LIN {X -0.135,Y -641.300,Z 780.617,A 0.000,B 0.000,C 90.000,E1 327.041} C_DIS
LIN {X 0.233,Y -645.781,Z 780.611,A 0.000,B 0.000,C 90.000,E1 326.008} C_DIS
LIN {X 0.128,Y -649.952,Z 780.606,A 0.000,B 0.000,C 90.000,E1 325.022} C_DIS
LIN {X 0.080,Y -653.850,Z 780.600,A 0.000,B 0.000,C 90.000,E1 324.036} C_DIS
LIN {X 0.081,Y -657.396,Z 780.595,A 0.000,B 0.000,C 90.000,E1 323.050} C_DIS
LIN {X 0.118,Y -660.884,Z 780.589,A 0.000,B 0.000,C 90.000,E1 322.065} C_DIS
LIN {X -0.359,Y -664.827,Z 780.583,A 0.000,B 0.000,C 90.000,E1 320.884} C_DIS
LIN {X -0.338,Y -667.859,Z 780.577,A 0.000,B 0.000,C 90.000,E1 319.908} C_DIS
LIN {X -0.271,Y -671.350,Z 780.570,A 0.000,B 0.000,C 90.000,E1 318.690} C_DIS
LIN {X -0.147,Y -674.584,Z 780.564,A 0.000,B 0.000,C 90.000,E1 317.472} C_DIS
LIN {X -0.008,Y -677.297,Z 780.557,A 0.000,B 0.000,C 90.000,E1 316.257} C_DIS
LIN {X -0.291,Y -679.717,Z 780.550,A 0.000,B 0.000,C 90.000,E1 315.081} C_DIS
LIN {X -0.066,Y -681.929,Z 780.544,A 0.000,B 0.000,C 90.000,E1 313.866} C_DIS
LIN {X -0.279,Y -683.940,Z 780.537,A 0.000,B 0.000,C 90.000,E1 312.690} C_DIS
LIN {X 0.049,Y -685.760,Z 780.530,A 0.000,B 0.000,C 90.000,E1 311.472} C_DIS
LIN {X -0.114,Y -687.422,Z 780.524,A 0.000,B 0.000,C 90.000,E1 310.297} C_DIS
LIN {X -0.180,Y -688.753,Z 780.517,A 0.000,B 0.000,C 90.000,E1 309.116} C_DIS
LIN {X -0.050,Y -690.190,Z 780.509,A 0.000,B 0.000,C 90.000,E1 307.684} C_DIS
LIN {X -0.124,Y -691.112,Z 780.504,A 0.000,B 0.000,C 90.000,E1 306.744} C_DIS
LIN {X 0.057,Y -692.345,Z 780.496,A 0.000,B 0.000,C 90.000,E1 305.311} C_DIS
LIN {X 0.205,Y -693.268,Z 780.490,A 0.000,B 0.000,C 90.000,E1 304.119} C_DIS
LIN {X 0.235,Y -694.476,Z 780.481,A 0.000,B 0.000,C 90.000,E1 302.467} C_DIS
LIN {X -0.090,Y -695.755,Z 780.471,A 0.000,B 0.000,C 90.000,E1 300.846} C_DIS
LIN {X 0.307,Y -696.373,Z 780.466,A 0.000,B 0.000,C 90.000,E1 299.873} C_DIS
LIN {X 0.018,Y -697.038,Z 780.458,A 0.000,B 0.000,C 90.000,E1 298.487} C_DIS
LIN {X -0.332,Y -697.783,Z 780.449,A 0.000,B 0.000,C 90.000,E1 296.873} C_DIS
LIN {X 0.192,Y -699.103,Z 780.437,A 0.000,B 0.000,C 90.000,E1 294.719} C_DIS
LIN {X 0.088,Y -699.011,Z 780.435,A 0.000,B 0.000,C 90.000,E1 294.259} C_DIS
LIN {X 0.067,Y -698.774,Z 780.434,A 0.000,B 0.000,C 90.000,E1 294.027} C_DIS
LIN {X -0.045,Y -697.662,Z 780.431,A 0.000,B 0.000,C 90.000,E1 293.567} C_DIS
LIN {X -0.062,Y -696.673,Z 780.430,A 0.000,B 0.000,C 90.000,E1 293.334} C_DIS
LIN {X 0.195,Y -694.685,Z 780.428,A 0.000,B 0.000,C 90.000,E1 293.078} C_DIS
LIN {X 0.174,Y -692.575,Z 780.427,A 0.000,B 0.000,C 90.000,E1 292.845} C_DIS
LIN {X -0.344,Y -691.398,Z 780.426,A 0.000,B 0.000,C 90.000,E1 292.770} C_DIS
LIN {X -0.222,Y -689.693,Z 780.426,A 0.000,B 0.000,C 90.000,E1 292.642} C_DIS
LIN {X 0.320,Y -683.390,Z 780.424,A 0.000,B 0.000,C 90.000,E1 292.333} C_DIS
LIN {X 0.365,Y -679.497,Z 780.424,A 0.000,B 0.000,C 90.000,E1 292.206} C_DIS
LIN {X 0.119,Y -673.718,Z 780.423,A 0.000,B 0.000,C 90.000,E1 292.078} C_DIS
LIN {X -0.079,Y -664.421,Z 780.422,A 0.000,B 0.000,C 90.000,E1 291.950} C_DIS
LIN {X 0.178,Y -654.094,Z 780.421,A 0.000,B 0.000,C 90.000,E1 291.770} C_DIS
LIN {X 0.001,Y -640.328,Z 780.420,A 0.000,B 0.000,C 90.000,E1 291.535} C_DIS
LIN {X 0.328,Y -616.048,Z 780.417,A 0.000,B 0.000,C 90.000,E1 290.972} C_DIS
LIN {X -0.071,Y -595.435,Z 780.414,A 0.000,B 0.000,C 90.000,E1 290.482} C_DIS
LIN {X -0.040,Y -571.555,Z 780.410,A 0.000,B 0.000,C 90.000,E1 289.758} C_DIS
LIN {X 0.063,Y -565.181,Z 780.409,A 0.000,B 0.000,C 90.000,E1 289.523} C_DIS
LIN {X 0.046,Y -560.669,Z 780.407,A 0.000,B 0.000,C 90.000,E1 289.322} C_DIS
LIN {X -0.169,Y -557.657,Z 780.406,A 0.000,B 0.000,C 90.000,E1 289.087} C_DIS
LIN {X -0.152,Y -556.753,Z 780.405,A 0.000,B 0.000,C 90.000,E1 288.906} C_DIS
LIN {X 0.258,Y -556.190,Z 780.404,A 0.000,B 0.000,C 90.000,E1 288.725} C_DIS
LIN {X -0.274,Y -555.270,Z 780.402,A 0.000,B 0.000,C 90.000,E1 288.362} C_DIS
LIN {X 0.220,Y -554.706,Z 780.399,A 0.000,B 0.000,C 90.000,E1 287.764} C_DIS
LIN {X -0.169,Y -554.398,Z 780.394,A 0.000,B 0.000,C 90.000,E1 286.968} C_DIS
LIN {X 0.001,Y -553.355,Z 780.382,A 0.000,B 0.000,C 90.000,E1 284.717} C_DIS
LIN {X -0.097,Y -552.709,Z 780.371,A 0.000,B 0.000,C 90.000,E1 282.771} C_DIS
LIN {X 0.209,Y -551.975,Z 780.360,A 0.000,B 0.000,C 90.000,E1 280.782} C_DIS
LIN {X 0.251,Y -551.570,Z 780.352,A 0.000,B 0.000,C 90.000,E1 279.378} C_DIS
LIN {X -0.222,Y -551.091,Z 780.341,A 0.000,B 0.000,C 90.000,E1 277.466} C_DIS
LIN {X -0.037,Y -550.765,Z 780.337,A 0.000,B 0.000,C 90.000,E1 276.606} C_DIS
LIN {X -0.194,Y -549.990,Z 780.329,A 0.000,B 0.000,C 90.000,E1 275.220} C_DIS
LIN {X 0.172,Y -548.872,Z 780.320,A 0.000,B 0.000,C 90.000,E1 273.498} C_DIS
LIN {X 0.007,Y -547.653,Z 780.309,A 0.000,B 0.000,C 90.000,E1 271.547} C_DIS
LIN {X 0.192,Y -546.992,Z 780.302,A 0.000,B 0.000,C 90.000,E1 270.401} C_DIS
LIN {X -0.093,Y -545.804,Z 780.293,A 0.000,B 0.000,C 90.000,E1 268.740} C_DIS
LIN {X 0.211,Y -544.440,Z 780.282,A 0.000,B 0.000,C 90.000,E1 266.731} C_DIS
LIN {X -0.058,Y -543.288,Z 780.271,A 0.000,B 0.000,C 90.000,E1 264.780} C_DIS
LIN {X 0.118,Y -542.505,Z 780.265,A 0.000,B 0.000,C 90.000,E1 263.628} C_DIS
LIN {X -0.188,Y -541.619,Z 780.258,A 0.000,B 0.000,C 90.000,E1 262.527} C_DIS
LIN {X 0.159,Y -539.693,Z 780.246,A 0.000,B 0.000,C 90.000,E1 260.218} C_DIS
LIN {X -0.021,Y -538.448,Z 780.238,A 0.000,B 0.000,C 90.000,E1 258.814} C_DIS
LIN {X -0.218,Y -537.131,Z 780.230,A 0.000,B 0.000,C 90.000,E1 257.409} C_DIS
LIN {X 0.204,Y -535.771,Z 780.222,A 0.000,B 0.000,C 90.000,E1 255.936} C_DIS
LIN {X 0.076,Y -534.243,Z 780.214,A 0.000,B 0.000,C 90.000,E1 254.519} C_DIS
LIN {X -0.040,Y -531.633,Z 780.201,A 0.000,B 0.000,C 90.000,E1 252.236} C_DIS
LIN {X 0.062,Y -529.928,Z 780.193,A 0.000,B 0.000,C 90.000,E1 250.786} C_DIS
LIN {X -0.057,Y -528.729,Z 780.189,A 0.000,B 0.000,C 90.000,E1 249.934} C_DIS
LIN {X -0.169,Y -525.843,Z 780.177,A 0.000,B 0.000,C 90.000,E1 247.922} C_DIS
LIN {X 0.025,Y -522.729,Z 780.166,A 0.000,B 0.000,C 90.000,E1 245.869} C_DIS
LIN {X 0.231,Y -521.360,Z 780.161,A 0.000,B 0.000,C 90.000,E1 244.973} C_DIS
LIN {X 0.044,Y -518.031,Z 780.150,A 0.000,B 0.000,C 90.000,E1 242.948} C_DIS
LIN {X 0.103,Y -515.939,Z 780.143,A 0.000,B 0.000,C 90.000,E1 241.769} C_DIS
LIN {X 0.136,Y -513.734,Z 780.137,A 0.000,B 0.000,C 90.000,E1 240.589} C_DIS
LIN {X 0.039,Y -510.898,Z 780.129,A 0.000,B 0.000,C 90.000,E1 239.125} C_DIS
LIN {X -0.012,Y -508.599,Z 780.122,A 0.000,B 0.000,C 90.000,E1 237.946} C_DIS
LIN {X 0.011,Y -506.111,Z 780.115,A 0.000,B 0.000,C 90.000,E1 236.755} C_DIS
LIN {X -0.165,Y -504.204,Z 780.110,A 0.000,B 0.000,C 90.000,E1 235.881} C_DIS
LIN {X -0.195,Y -501.477,Z 780.104,A 0.000,B 0.000,C 90.000,E1 234.689} C_DIS
LIN {X -0.267,Y -498.555,Z 780.097,A 0.000,B 0.000,C 90.000,E1 233.497} C_DIS
LIN {X -0.224,Y -494.759,Z 780.089,A 0.000,B 0.000,C 90.000,E1 231.984} C_DIS
LIN {X -0.103,Y -490.281,Z 780.079,A 0.000,B 0.000,C 90.000,E1 230.150} C_DIS
LIN {X -0.037,Y -484.029,Z 780.063,A 0.000,B 0.000,C 90.000,E1 227.391} C_DIS
LIN {X 0.308,Y -480.729,Z 780.055,A 0.000,B 0.000,C 90.000,E1 225.810} C_DIS
LIN {X -0.314,Y -476.642,Z 780.044,A 0.000,B 0.000,C 90.000,E1 224.028} C_DIS
LIN {X -0.110,Y -473.271,Z 780.036,A 0.000,B 0.000,C 90.000,E1 222.447} C_DIS
LIN {X 0.139,Y -469.135,Z 780.025,A 0.000,B 0.000,C 90.000,E1 220.539} C_DIS
LIN {X -0.014,Y -465.253,Z 780.015,A 0.000,B 0.000,C 90.000,E1 218.669} C_DIS
LIN {X -0.049,Y -459.917,Z 780.001,A 0.000,B 0.000,C 90.000,E1 216.137} C_DIS
LIN {X 0.133,Y -455.957,Z 779.990,A 0.000,B 0.000,C 90.000,E1 214.199} C_DIS
LIN {X 0.074,Y -451.441,Z 779.978,A 0.000,B 0.000,C 90.000,E1 211.957} C_DIS
LIN {X 0.120,Y -448.322,Z 779.969,A 0.000,B 0.000,C 90.000,E1 210.335} C_DIS
LIN {X -0.129,Y -445.213,Z 779.960,A 0.000,B 0.000,C 90.000,E1 208.743} C_DIS
LIN {X 0.132,Y -442.126,Z 779.951,A 0.000,B 0.000,C 90.000,E1 207.078} C_DIS
LIN {X -0.058,Y -438.986,Z 779.941,A 0.000,B 0.000,C 90.000,E1 205.463} C_DIS
LIN {X -0.111,Y -435.916,Z 779.932,A 0.000,B 0.000,C 90.000,E1 203.823} C_DIS
LIN {X 0.003,Y -432.784,Z 779.923,A 0.000,B 0.000,C 90.000,E1 202.153} C_DIS
LIN {X 0.243,Y -430.223,Z 779.916,A 0.000,B 0.000,C 90.000,E1 200.791} C_DIS
LIN {X -0.052,Y -425.741,Z 779.903,A 0.000,B 0.000,C 90.000,E1 198.489} C_DIS
LIN {X -0.025,Y -422.562,Z 779.893,A 0.000,B 0.000,C 90.000,E1 196.804} C_DIS
LIN {X -0.183,Y -419.202,Z 779.884,A 0.000,B 0.000,C 90.000,E1 195.134} C_DIS
LIN {X 0.087,Y -414.754,Z 779.871,A 0.000,B 0.000,C 90.000,E1 192.715} C_DIS
LIN {X 0.062,Y -411.612,Z 779.861,A 0.000,B 0.000,C 90.000,E1 191.007} C_DIS
LIN {X -0.145,Y -407.322,Z 779.848,A 0.000,B 0.000,C 90.000,E1 188.624} C_DIS
LIN {X -0.144,Y -405.096,Z 779.840,A 0.000,B 0.000,C 90.000,E1 187.239} C_DIS
LIN {X 0.178,Y -402.144,Z 779.831,A 0.000,B 0.000,C 90.000,E1 185.454} C_DIS
LIN {X 0.078,Y -395.784,Z 779.807,A 0.000,B 0.000,C 90.000,E1 181.260} C_DIS
LIN {X 0.077,Y -393.265,Z 779.795,A 0.000,B 0.000,C 90.000,E1 179.141} C_DIS
LIN {X -0.127,Y -390.209,Z 779.780,A 0.000,B 0.000,C 90.000,E1 176.331} C_DIS
LIN {X -0.108,Y -388.525,Z 779.770,A 0.000,B 0.000,C 90.000,E1 174.546} C_DIS
LIN {X 0.128,Y -386.230,Z 779.756,A 0.000,B 0.000,C 90.000,E1 172.008} C_DIS
LIN {X 0.022,Y -384.179,Z 779.742,A 0.000,B 0.000,C 90.000,E1 169.511} C_DIS
LIN {X 0.000,Y -382.678,Z 779.730,A 0.000,B 0.000,C 90.000,E1 167.353} C_DIS
LIN {X 0.105,Y -381.329,Z 779.716,A 0.000,B 0.000,C 90.000,E1 164.810} C_DIS
LIN {X 0.012,Y -380.680,Z 779.708,A 0.000,B 0.000,C 90.000,E1 163.378} C_DIS
LIN {X 0.027,Y -379.601,Z 779.690,A 0.000,B 0.000,C 90.000,E1 160.115} C_DIS
LIN {X -0.068,Y -379.365,Z 779.661,A 0.000,B 0.000,C 90.000,E1 155.049} C_DIS
LIN {X -0.006,Y -380.951,Z 779.639,A 0.000,B 0.000,C 90.000,E1 151.051} C_DIS
LIN {X -0.102,Y -383.270,Z 779.625,A 0.000,B 0.000,C 90.000,E1 148.535} C_DIS
LIN {X -0.105,Y -384.702,Z 779.619,A 0.000,B 0.000,C 90.000,E1 147.454} C_DIS
LIN {X -0.161,Y -388.401,Z 779.607,A 0.000,B 0.000,C 90.000,E1 145.308} C_DIS
LIN {X 0.051,Y -390.026,Z 779.603,A 0.000,B 0.000,C 90.000,E1 144.562} C_DIS
LIN {X -0.046,Y -392.045,Z 779.599,A 0.000,B 0.000,C 90.000,E1 143.863} C_DIS
LIN {X 0.108,Y -394.435,Z 779.595,A 0.000,B 0.000,C 90.000,E1 143.130} C_DIS
LIN {X 0.179,Y -397.031,Z 779.592,A 0.000,B 0.000,C 90.000,E1 142.477} C_DIS
LIN {X 0.041,Y -399.851,Z 779.588,A 0.000,B 0.000,C 90.000,E1 141.904} C_DIS
LIN {X 0.055,Y -402.995,Z 779.586,A 0.000,B 0.000,C 90.000,E1 141.376} C_DIS
LIN {X -0.179,Y -407.195,Z 779.582,A 0.000,B 0.000,C 90.000,E1 140.803} C_DIS
LIN {X -0.022,Y -422.989,Z 779.572,A 0.000,B 0.000,C 90.000,E1 138.895} C_DIS
LIN {X -0.088,Y -439.732,Z 779.561,A 0.000,B 0.000,C 90.000,E1 137.067} C_DIS
LIN {X 0.241,Y -449.355,Z 779.556,A 0.000,B 0.000,C 90.000,E1 135.972} C_DIS
LIN {X 0.037,Y -458.769,Z 779.550,A 0.000,B 0.000,C 90.000,E1 134.919} C_DIS
LIN {X 0.196,Y -465.141,Z 779.545,A 0.000,B 0.000,C 90.000,E1 134.109} C_DIS
LIN {X -0.046,Y -473.687,Z 779.539,A 0.000,B 0.000,C 90.000,E1 133.056} C_DIS
LIN {X -0.070,Y -480.870,Z 779.534,A 0.000,B 0.000,C 90.000,E1 132.123} C_DIS
LIN {X -0.026,Y -486.422,Z 779.530,A 0.000,B 0.000,C 90.000,E1 131.353} C_DIS
LIN {X -0.229,Y -492.767,Z 779.525,A 0.000,B 0.000,C 90.000,E1 130.458} C_DIS
LIN {X 0.252,Y -497.825,Z 779.520,A 0.000,B 0.000,C 90.000,E1 129.644} C_DIS
LIN {X -0.013,Y -501.651,Z 779.517,A 0.000,B 0.000,C 90.000,E1 129.072} C_DIS
LIN {X -0.147,Y -508.748,Z 779.510,A 0.000,B 0.000,C 90.000,E1 127.890} C_DIS
LIN {X -0.221,Y -512.922,Z 779.506,A 0.000,B 0.000,C 90.000,E1 127.156} C_DIS
LIN {X -0.032,Y -517.651,Z 779.501,A 0.000,B 0.000,C 90.000,E1 126.251} C_DIS
LIN {X -0.079,Y -522.953,Z 779.496,A 0.000,B 0.000,C 90.000,E1 125.231} C_DIS
LIN {X 0.263,Y -525.864,Z 779.492,A 0.000,B 0.000,C 90.000,E1 124.612} C_DIS
LIN {X 0.061,Y -527.701,Z 779.490,A 0.000,B 0.000,C 90.000,E1 124.199} C_DIS
LIN {X -0.095,Y -530.217,Z 779.487,A 0.000,B 0.000,C 90.000,E1 123.658} C_DIS
LIN {X 0.293,Y -533.847,Z 779.482,A 0.000,B 0.000,C 90.000,E1 122.752} C_DIS
LIN {X -0.317,Y -538.451,Z 779.476,A 0.000,B 0.000,C 90.000,E1 121.671} C_DIS
LIN {X -0.133,Y -541.646,Z 779.471,A 0.000,B 0.000,C 90.000,E1 120.797} C_DIS
LIN {X 0.084,Y -544.591,Z 779.466,A 0.000,B 0.000,C 90.000,E1 119.922} C_DIS
LIN {X -0.187,Y -548.316,Z 779.460,A 0.000,B 0.000,C 90.000,E1 118.821} C_DIS
LIN {X -0.165,Y -550.955,Z 779.455,A 0.000,B 0.000,C 90.000,E1 117.975} C_DIS
LIN {X -0.116,Y -553.416,Z 779.451,A 0.000,B 0.000,C 90.000,E1 117.129} C_DIS
LIN {X -0.046,Y -555.467,Z 779.446,A 0.000,B 0.000,C 90.000,E1 116.283} C_DIS
LIN {X -0.200,Y -557.174,Z 779.441,A 0.000,B 0.000,C 90.000,E1 115.463} C_DIS
LIN {X 0.174,Y -558.623,Z 779.437,A 0.000,B 0.000,C 90.000,E1 114.591} C_DIS
LIN {X 0.057,Y -559.762,Z 779.432,A 0.000,B 0.000,C 90.000,E1 113.770} C_DIS
LIN {X -0.052,Y -561.988,Z 779.421,A 0.000,B 0.000,C 90.000,E1 111.844} C_DIS
LIN {X -0.032,Y -563.169,Z 779.415,A 0.000,B 0.000,C 90.000,E1 110.737} C_DIS
LIN {X 0.138,Y -564.459,Z 779.408,A 0.000,B 0.000,C 90.000,E1 109.341} C_DIS
LIN {X 0.182,Y -565.400,Z 779.401,A 0.000,B 0.000,C 90.000,E1 108.236} C_DIS
LIN {X -0.174,Y -566.633,Z 779.392,A 0.000,B 0.000,C 90.000,E1 106.622} C_DIS
LIN {X 0.044,Y -567.863,Z 779.383,A 0.000,B 0.000,C 90.000,E1 104.954} C_DIS
LIN {X -0.230,Y -569.434,Z 779.372,A 0.000,B 0.000,C 90.000,E1 103.063} C_DIS
LIN {X -0.038,Y -571.056,Z 779.362,A 0.000,B 0.000,C 90.000,E1 101.130} C_DIS
LIN {X -0.207,Y -572.206,Z 779.354,A 0.000,B 0.000,C 90.000,E1 99.782} C_DIS
LIN {X -0.094,Y -573.128,Z 779.348,A 0.000,B 0.000,C 90.000,E1 98.681} C_DIS
LIN {X -0.046,Y -574.003,Z 779.342,A 0.000,B 0.000,C 90.000,E1 97.587} C_DIS
LIN {X 0.222,Y -574.957,Z 779.335,A 0.000,B 0.000,C 90.000,E1 96.201} C_DIS
LIN {X 0.061,Y -575.957,Z 779.326,A 0.000,B 0.000,C 90.000,E1 94.588} C_DIS
LIN {X 0.261,Y -576.753,Z 779.318,A 0.000,B 0.000,C 90.000,E1 93.212} C_DIS
LIN {X -0.092,Y -577.477,Z 779.310,A 0.000,B 0.000,C 90.000,E1 91.892} C_DIS
LIN {X 0.136,Y -578.083,Z 779.303,A 0.000,B 0.000,C 90.000,E1 90.516} C_DIS
LIN {X -0.214,Y -578.652,Z 779.295,A 0.000,B 0.000,C 90.000,E1 89.198} C_DIS
LIN {X 0.198,Y -579.213,Z 779.286,A 0.000,B 0.000,C 90.000,E1 87.535} C_DIS
LIN {X 0.077,Y -579.648,Z 779.277,A 0.000,B 0.000,C 90.000,E1 85.927} C_DIS
LIN {X -0.245,Y -579.935,Z 779.270,A 0.000,B 0.000,C 90.000,E1 84.609} C_DIS
LIN {X 0.118,Y -580.126,Z 779.262,A 0.000,B 0.000,C 90.000,E1 83.223} C_DIS
LIN {X 0.137,Y -580.396,Z 779.253,A 0.000,B 0.000,C 90.000,E1 81.602} C_DIS
LIN {X -0.189,Y -580.544,Z 779.243,A 0.000,B 0.000,C 90.000,E1 79.746} C_DIS
LIN {X -0.304,Y -580.525,Z 779.235,A 0.000,B 0.000,C 90.000,E1 78.409} C_DIS
LIN {X 0.048,Y -580.361,Z 779.227,A 0.000,B 0.000,C 90.000,E1 76.756} C_DIS
LIN {X -0.301,Y -579.964,Z 779.218,A 0.000,B 0.000,C 90.000,E1 75.172} C_DIS
LIN {X 0.160,Y -579.646,Z 779.211,A 0.000,B 0.000,C 90.000,E1 74.047} C_DIS
LIN {X -0.123,Y -579.271,Z 779.204,A 0.000,B 0.000,C 90.000,E1 72.725} C_DIS
LIN {X 0.139,Y -578.726,Z 779.197,A 0.000,B 0.000,C 90.000,E1 71.348} C_DIS
LIN {X -0.134,Y -577.937,Z 779.188,A 0.000,B 0.000,C 90.000,E1 69.752} C_DIS
LIN {X 0.123,Y -577.021,Z 779.178,A 0.000,B 0.000,C 90.000,E1 68.103} C_DIS
LIN {X 0.191,Y -576.061,Z 779.171,A 0.000,B 0.000,C 90.000,E1 66.741} C_DIS
LIN {X -0.054,Y -574.990,Z 779.163,A 0.000,B 0.000,C 90.000,E1 65.409} C_DIS
LIN {X -0.151,Y -573.984,Z 779.157,A 0.000,B 0.000,C 90.000,E1 64.332} C_DIS
LIN {X -0.267,Y -572.836,Z 779.151,A 0.000,B 0.000,C 90.000,E1 63.256} C_DIS
LIN {X -0.141,Y -571.424,Z 779.145,A 0.000,B 0.000,C 90.000,E1 62.153} C_DIS
LIN {X -0.037,Y -569.901,Z 779.139,A 0.000,B 0.000,C 90.000,E1 61.051} C_DIS
LIN {X 0.142,Y -567.556,Z 779.132,A 0.000,B 0.000,C 90.000,E1 59.665} C_DIS
LIN {X -0.018,Y -565.426,Z 779.125,A 0.000,B 0.000,C 90.000,E1 58.584} C_DIS
LIN {X 0.172,Y -563.573,Z 779.121,A 0.000,B 0.000,C 90.000,E1 57.740} C_DIS
LIN {X 0.162,Y -561.585,Z 779.116,A 0.000,B 0.000,C 90.000,E1 56.914} C_DIS
LIN {X 0.221,Y -558.486,Z 779.110,A 0.000,B 0.000,C 90.000,E1 55.801} C_DIS
LIN {X 0.077,Y -556.874,Z 779.107,A 0.000,B 0.000,C 90.000,E1 55.261} C_DIS
LIN {X 0.316,Y -554.145,Z 779.102,A 0.000,B 0.000,C 90.000,E1 54.402} C_DIS
LIN {X 0.135,Y -552.254,Z 779.099,A 0.000,B 0.000,C 90.000,E1 53.863} C_DIS
LIN {X -0.116,Y -549.048,Z 779.095,A 0.000,B 0.000,C 90.000,E1 53.050} C_DIS
LIN {X 0.042,Y -545.428,Z 779.090,A 0.000,B 0.000,C 90.000,E1 52.190} C_DIS
LIN {X 0.303,Y -542.119,Z 779.086,A 0.000,B 0.000,C 90.000,E1 51.457} C_DIS
LIN {X -0.067,Y -539.301,Z 779.083,A 0.000,B 0.000,C 90.000,E1 50.928} C_DIS
LIN {X -0.036,Y -536.250,Z 779.080,A 0.000,B 0.000,C 90.000,E1 50.356} C_DIS
LIN {X 0.136,Y -531.961,Z 779.076,A 0.000,B 0.000,C 90.000,E1 49.622} C_DIS
LIN {X 0.048,Y -528.167,Z 779.073,A 0.000,B 0.000,C 90.000,E1 49.057} C_DIS
LIN {X -0.014,Y -523.886,Z 779.069,A 0.000,B 0.000,C 90.000,E1 48.485} C_DIS
LIN {X 0.088,Y -520.380,Z 779.067,A 0.000,B 0.000,C 90.000,E1 48.038} C_DIS
LIN {X -0.292,Y -514.259,Z 779.063,A 0.000,B 0.000,C 90.000,E1 47.391} C_DIS
LIN {X 0.103,Y -508.775,Z 779.060,A 0.000,B 0.000,C 90.000,E1 46.782} C_DIS
LIN {X 0.049,Y -504.504,Z 779.058,A 0.000,B 0.000,C 90.000,E1 46.377} C_DIS
LIN {X -0.270,Y -498.499,Z 779.055,A 0.000,B 0.000,C 90.000,E1 45.891} C_DIS
LIN {X 0.047,Y -490.959,Z 779.051,A 0.000,B 0.000,C 90.000,E1 45.243} C_DIS
LIN {X -0.198,Y -482.988,Z 779.048,A 0.000,B 0.000,C 90.000,E1 44.676} C_DIS
LIN {X -0.031,Y -478.192,Z 779.046,A 0.000,B 0.000,C 90.000,E1 44.312} C_DIS
LIN {X -0.218,Y -465.311,Z 779.041,A 0.000,B 0.000,C 90.000,E1 43.461} C_DIS
LIN {X -0.052,Y -447.509,Z 779.035,A 0.000,B 0.000,C 90.000,E1 42.243} C_DIS
LIN {X -0.038,Y -423.711,Z 779.025,A 0.000,B 0.000,C 90.000,E1 40.539} C_DIS
LIN {X -0.085,Y -414.350,Z 779.021,A 0.000,B 0.000,C 90.000,E1 39.806} C_DIS
LIN {X -0.121,Y -410.052,Z 779.019,A 0.000,B 0.000,C 90.000,E1 39.439} C_DIS
LIN {X -0.064,Y -406.881,Z 779.017,A 0.000,B 0.000,C 90.000,E1 39.116} C_DIS
LIN {X -0.090,Y -406.862,Z 779.017,A 0.000,B 0.000,C 90.000,E1 39.116} C_DIS
LIN {X -0.144,Y -405.592,Z 779.013,A 0.000,B 0.000,C 90.000,E1 38.382} C_DIS
LIN {X -0.178,Y -397.338,Z 778.990,A 0.000,B 0.000,C 90.000,E1 34.199} C_DIS
LIN {X -0.099,Y -398.170,Z 778.970,A 0.000,B 0.000,C 90.000,E1 30.669} C_DIS
LIN {X -0.014,Y -399.475,Z 778.955,A 0.000,B 0.000,C 90.000,E1 27.847} C_DIS
LIN {X -0.143,Y -400.907,Z 778.941,A 0.000,B 0.000,C 90.000,E1 25.412} C_DIS
LIN {X -0.002,Y -403.446,Z 778.922,A 0.000,B 0.000,C 90.000,E1 21.897} C_DIS
LIN {X 0.237,Y -407.649,Z 778.898,A 0.000,B 0.000,C 90.000,E1 17.692} C_DIS
LIN {X 0.064,Y -411.401,Z 778.883,A 0.000,B 0.000,C 90.000,E1 14.954} C_DIS
LIN {X 0.175,Y -415.134,Z 778.870,A 0.000,B 0.000,C 90.000,E1 12.535} C_DIS
LIN {X 0.157,Y -418.602,Z 778.858,A 0.000,B 0.000,C 90.000,E1 10.489} C_DIS
LIN {X 0.146,Y -422.105,Z 778.847,A 0.000,B 0.000,C 90.000,E1 8.454} C_DIS
LIN {X -0.018,Y -424.473,Z 778.840,A 0.000,B 0.000,C 90.000,E1 7.125} C_DIS
LIN {X 0.079,Y -428.564,Z 778.827,A 0.000,B 0.000,C 90.000,E1 4.759} C_DIS
LIN {X -0.065,Y -431.053,Z 778.819,A 0.000,B 0.000,C 90.000,E1 3.440} C_DIS
LIN {X 0.115,Y -435.530,Z 778.806,A 0.000,B 0.000,C 90.000,E1 1.088} C_DIS
LIN {X 0.166,Y -440.867,Z 778.792,A 0.000,B 0.000,C 90.000,E1 358.453} C_DIS
LIN {X 0.035,Y -447.459,Z 778.775,A 0.000,B 0.000,C 90.000,E1 355.527} C_DIS
LIN {X -0.034,Y -451.280,Z 778.766,A 0.000,B 0.000,C 90.000,E1 353.913} C_DIS
LIN {X 0.185,Y -455.829,Z 778.755,A 0.000,B 0.000,C 90.000,E1 351.951} C_DIS
LIN {X -0.116,Y -459.532,Z 778.747,A 0.000,B 0.000,C 90.000,E1 350.387} C_DIS
LIN {X -0.068,Y -462.375,Z 778.740,A 0.000,B 0.000,C 90.000,E1 349.106} C_DIS
LIN {X 0.020,Y -465.229,Z 778.732,A 0.000,B 0.000,C 90.000,E1 347.825} C_DIS
LIN {X -0.015,Y -467.907,Z 778.727,A 0.000,B 0.000,C 90.000,E1 346.881} C_DIS
LIN {X -0.018,Y -469.717,Z 778.725,A 0.000,B 0.000,C 90.000,E1 346.408} C_DIS
LIN {X 0.143,Y -471.675,Z 778.722,A 0.000,B 0.000,C 90.000,E1 345.992} C_DIS
LIN {X 0.164,Y -474.732,Z 778.720,A 0.000,B 0.000,C 90.000,E1 345.519} C_DIS
LIN {X 0.071,Y -477.727,Z 778.718,A 0.000,B 0.000,C 90.000,E1 345.172} C_DIS
LIN {X 0.191,Y -484.333,Z 778.714,A 0.000,B 0.000,C 90.000,E1 344.519} C_DIS
LIN {X -0.038,Y -494.816,Z 778.710,A 0.000,B 0.000,C 90.000,E1 343.740} C_DIS
LIN {X 0.106,Y -505.698,Z 778.705,A 0.000,B 0.000,C 90.000,E1 342.960} C_DIS
LIN {X 0.244,Y -531.163,Z 778.696,A 0.000,B 0.000,C 90.000,E1 341.275} C_DIS
LIN {X 0.086,Y -540.472,Z 778.693,A 0.000,B 0.000,C 90.000,E1 340.678} C_DIS
LIN {X -0.131,Y -547.904,Z 778.690,A 0.000,B 0.000,C 90.000,E1 340.188} C_DIS
LIN {X 0.013,Y -553.282,Z 778.688,A 0.000,B 0.000,C 90.000,E1 339.752} C_DIS
LIN {X 0.120,Y -558.763,Z 778.685,A 0.000,B 0.000,C 90.000,E1 339.263} C_DIS
LIN {X -0.056,Y -564.082,Z 778.682,A 0.000,B 0.000,C 90.000,E1 338.773} C_DIS
LIN {X 0.059,Y -569.107,Z 778.679,A 0.000,B 0.000,C 90.000,E1 338.230} C_DIS
LIN {X -0.154,Y -573.863,Z 778.676,A 0.000,B 0.000,C 90.000,E1 337.720} C_DIS
LIN {X -0.174,Y -578.430,Z 778.673,A 0.000,B 0.000,C 90.000,E1 337.177} C_DIS
LIN {X -0.207,Y -586.708,Z 778.667,A 0.000,B 0.000,C 90.000,E1 336.102} C_DIS
LIN {X 0.040,Y -591.583,Z 778.663,A 0.000,B 0.000,C 90.000,E1 335.409} C_DIS
LIN {X 0.287,Y -597.165,Z 778.659,A 0.000,B 0.000,C 90.000,E1 334.588} C_DIS
LIN {X -0.013,Y -604.187,Z 778.653,A 0.000,B 0.000,C 90.000,E1 333.563} C_DIS
LIN {X -0.203,Y -609.951,Z 778.648,A 0.000,B 0.000,C 90.000,E1 332.666} C_DIS
LIN {X -0.343,Y -616.269,Z 778.642,A 0.000,B 0.000,C 90.000,E1 331.641} C_DIS
LIN {X -0.099,Y -620.772,Z 778.638,A 0.000,B 0.000,C 90.000,E1 330.845} C_DIS
LIN {X 0.208,Y -627.309,Z 778.632,A 0.000,B 0.000,C 90.000,E1 329.665} C_DIS
LIN {X 0.034,Y -631.469,Z 778.627,A 0.000,B 0.000,C 90.000,E1 328.918} C_DIS
LIN {X -0.080,Y -635.974,Z 778.622,A 0.000,B 0.000,C 90.000,E1 328.043} C_DIS
LIN {X -0.088,Y -641.838,Z 778.615,A 0.000,B 0.000,C 90.000,E1 326.786} C_DIS
LIN {X -0.254,Y -646.324,Z 778.610,A 0.000,B 0.000,C 90.000,E1 325.801} C_DIS
LIN {X 0.176,Y -650.529,Z 778.604,A 0.000,B 0.000,C 90.000,E1 324.769} C_DIS
LIN {X 0.129,Y -654.395,Z 778.599,A 0.000,B 0.000,C 90.000,E1 323.783} C_DIS
LIN {X 0.019,Y -659.702,Z 778.591,A 0.000,B 0.000,C 90.000,E1 322.316} C_DIS
LIN {X 0.083,Y -662.981,Z 778.585,A 0.000,B 0.000,C 90.000,E1 321.331} C_DIS
LIN {X 0.081,Y -666.115,Z 778.580,A 0.000,B 0.000,C 90.000,E1 320.356} C_DIS
LIN {X 0.128,Y -668.352,Z 778.576,A 0.000,B 0.000,C 90.000,E1 319.622} C_DIS
LIN {X -0.310,Y -671.198,Z 778.570,A 0.000,B 0.000,C 90.000,E1 318.690} C_DIS
LIN {X -0.208,Y -673.865,Z 778.565,A 0.000,B 0.000,C 90.000,E1 317.715} C_DIS
LIN {X -0.084,Y -676.699,Z 778.558,A 0.000,B 0.000,C 90.000,E1 316.500} C_DIS
LIN {X 0.034,Y -678.248,Z 778.554,A 0.000,B 0.000,C 90.000,E1 315.769} C_DIS
LIN {X -0.293,Y -680.168,Z 778.549,A 0.000,B 0.000,C 90.000,E1 314.838} C_DIS
LIN {X -0.110,Y -681.960,Z 778.544,A 0.000,B 0.000,C 90.000,E1 313.866} C_DIS
LIN {X -0.323,Y -684.043,Z 778.537,A 0.000,B 0.000,C 90.000,E1 312.690} C_DIS
LIN {X 0.404,Y -685.542,Z 778.532,A 0.000,B 0.000,C 90.000,E1 311.676} C_DIS
LIN {X -0.213,Y -687.235,Z 778.525,A 0.000,B 0.000,C 90.000,E1 310.539} C_DIS
LIN {X 0.103,Y -688.366,Z 778.520,A 0.000,B 0.000,C 90.000,E1 309.564} C_DIS
LIN {X -0.317,Y -689.896,Z 778.512,A 0.000,B 0.000,C 90.000,E1 308.177} C_DIS
LIN {X 0.205,Y -691.082,Z 778.505,A 0.000,B 0.000,C 90.000,E1 306.950} C_DIS
LIN {X 0.384,Y -692.332,Z 778.498,A 0.000,B 0.000,C 90.000,E1 305.518} C_DIS
LIN {X -0.431,Y -693.272,Z 778.491,A 0.000,B 0.000,C 90.000,E1 304.405} C_DIS
LIN {X 0.210,Y -694.653,Z 778.481,A 0.000,B 0.000,C 90.000,E1 302.467} C_DIS
LIN {X -0.110,Y -695.954,Z 778.471,A 0.000,B 0.000,C 90.000,E1 300.846} C_DIS
LIN {X -0.061,Y -696.665,Z 778.465,A 0.000,B 0.000,C 90.000,E1 299.667} C_DIS
LIN {X 0.264,Y -697.278,Z 778.457,A 0.000,B 0.000,C 90.000,E1 298.231} C_DIS
LIN {X 0.185,Y -698.182,Z 778.447,A 0.000,B 0.000,C 90.000,E1 296.360} C_DIS
LIN {X 0.186,Y -699.217,Z 778.437,A 0.000,B 0.000,C 90.000,E1 294.719} C_DIS
LIN {X 0.082,Y -699.097,Z 778.435,A 0.000,B 0.000,C 90.000,E1 294.259} C_DIS
LIN {X 0.061,Y -698.867,Z 778.434,A 0.000,B 0.000,C 90.000,E1 294.027} C_DIS
LIN {X -0.050,Y -697.661,Z 778.431,A 0.000,B 0.000,C 90.000,E1 293.567} C_DIS
LIN {X -0.067,Y -696.670,Z 778.430,A 0.000,B 0.000,C 90.000,E1 293.334} C_DIS
LIN {X 0.190,Y -694.681,Z 778.428,A 0.000,B 0.000,C 90.000,E1 293.078} C_DIS
LIN {X 0.168,Y -692.434,Z 778.427,A 0.000,B 0.000,C 90.000,E1 292.845} C_DIS
LIN {X -0.340,Y -691.200,Z 778.426,A 0.000,B 0.000,C 90.000,E1 292.770} C_DIS
LIN {X -0.210,Y -689.475,Z 778.426,A 0.000,B 0.000,C 90.000,E1 292.642} C_DIS
LIN {X 0.355,Y -683.125,Z 778.424,A 0.000,B 0.000,C 90.000,E1 292.333} C_DIS
LIN {X -0.191,Y -677.138,Z 778.423,A 0.000,B 0.000,C 90.000,E1 292.206} C_DIS
LIN {X 0.230,Y -673.195,Z 778.423,A 0.000,B 0.000,C 90.000,E1 292.078} C_DIS
LIN {X -0.090,Y -664.542,Z 778.422,A 0.000,B 0.000,C 90.000,E1 291.972} C_DIS
LIN {X 0.175,Y -657.248,Z 778.422,A 0.000,B 0.000,C 90.000,E1 291.844} C_DIS
LIN {X 0.380,Y -643.641,Z 778.420,A 0.000,B 0.000,C 90.000,E1 291.589} C_DIS
LIN {X 0.145,Y -633.655,Z 778.419,A 0.000,B 0.000,C 90.000,E1 291.408} C_DIS
LIN {X -0.207,Y -616.156,Z 778.417,A 0.000,B 0.000,C 90.000,E1 291.046} C_DIS
LIN {X -0.277,Y -592.089,Z 778.413,A 0.000,B 0.000,C 90.000,E1 290.429} C_DIS
LIN {X -0.148,Y -568.189,Z 778.409,A 0.000,B 0.000,C 90.000,E1 289.685} C_DIS
LIN {X -0.148,Y -565.212,Z 778.409,A 0.000,B 0.000,C 90.000,E1 289.577} C_DIS
LIN {X 0.282,Y -560.407,Z 778.408,A 0.000,B 0.000,C 90.000,E1 289.322} C_DIS
LIN {X 0.082,Y -557.446,Z 778.406,A 0.000,B 0.000,C 90.000,E1 289.087} C_DIS
LIN {X -0.087,Y -556.446,Z 778.405,A 0.000,B 0.000,C 90.000,E1 288.906} C_DIS
LIN {X 0.185,Y -555.685,Z 778.404,A 0.000,B 0.000,C 90.000,E1 288.598} C_DIS
LIN {X 0.132,Y -554.942,Z 778.400,A 0.000,B 0.000,C 90.000,E1 288.055} C_DIS
LIN {X -0.146,Y -554.456,Z 778.394,A 0.000,B 0.000,C 90.000,E1 286.968} C_DIS
LIN {X 0.025,Y -553.386,Z 778.382,A 0.000,B 0.000,C 90.000,E1 284.717} C_DIS
LIN {X -0.192,Y -552.810,Z 778.372,A 0.000,B 0.000,C 90.000,E1 283.063} C_DIS
LIN {X -0.007,Y -552.218,Z 778.363,A 0.000,B 0.000,C 90.000,E1 281.366} C_DIS
LIN {X 0.277,Y -551.603,Z 778.352,A 0.000,B 0.000,C 90.000,E1 279.378} C_DIS
LIN {X -0.196,Y -551.092,Z 778.341,A 0.000,B 0.000,C 90.000,E1 277.466} C_DIS
LIN {X -0.011,Y -550.766,Z 778.337,A 0.000,B 0.000,C 90.000,E1 276.606} C_DIS
LIN {X -0.168,Y -549.985,Z 778.329,A 0.000,B 0.000,C 90.000,E1 275.220} C_DIS
LIN {X 0.198,Y -548.843,Z 778.320,A 0.000,B 0.000,C 90.000,E1 273.498} C_DIS
LIN {X 0.033,Y -547.658,Z 778.309,A 0.000,B 0.000,C 90.000,E1 271.547} C_DIS
LIN {X 0.217,Y -546.967,Z 778.302,A 0.000,B 0.000,C 90.000,E1 270.401} C_DIS
LIN {X -0.067,Y -545.806,Z 778.293,A 0.000,B 0.000,C 90.000,E1 268.740} C_DIS
LIN {X 0.238,Y -544.469,Z 778.282,A 0.000,B 0.000,C 90.000,E1 266.731} C_DIS
LIN {X -0.032,Y -543.289,Z 778.271,A 0.000,B 0.000,C 90.000,E1 264.780} C_DIS
LIN {X 0.218,Y -542.319,Z 778.263,A 0.000,B 0.000,C 90.000,E1 263.337} C_DIS
LIN {X -0.161,Y -541.623,Z 778.258,A 0.000,B 0.000,C 90.000,E1 262.527} C_DIS
LIN {X 0.186,Y -539.718,Z 778.246,A 0.000,B 0.000,C 90.000,E1 260.218} C_DIS
LIN {X 0.006,Y -538.461,Z 778.238,A 0.000,B 0.000,C 90.000,E1 258.814} C_DIS
LIN {X -0.190,Y -537.166,Z 778.230,A 0.000,B 0.000,C 90.000,E1 257.409} C_DIS
LIN {X 0.232,Y -535.826,Z 778.222,A 0.000,B 0.000,C 90.000,E1 255.936} C_DIS
LIN {X 0.293,Y -533.928,Z 778.213,A 0.000,B 0.000,C 90.000,E1 254.212} C_DIS
LIN {X -0.200,Y -532.005,Z 778.203,A 0.000,B 0.000,C 90.000,E1 252.543} C_DIS
LIN {X -0.095,Y -530.348,Z 778.195,A 0.000,B 0.000,C 90.000,E1 251.094} C_DIS
LIN {X -0.026,Y -528.761,Z 778.189,A 0.000,B 0.000,C 90.000,E1 249.934} C_DIS
LIN {X -0.115,Y -526.302,Z 778.179,A 0.000,B 0.000,C 90.000,E1 248.209} C_DIS
LIN {X -0.113,Y -524.552,Z 778.172,A 0.000,B 0.000,C 90.000,E1 247.050} C_DIS
LIN {X -0.262,Y -522.376,Z 778.164,A 0.000,B 0.000,C 90.000,E1 245.613} C_DIS
LIN {X -0.233,Y -519.963,Z 778.156,A 0.000,B 0.000,C 90.000,E1 244.152} C_DIS
LIN {X -0.015,Y -517.566,Z 778.148,A 0.000,B 0.000,C 90.000,E1 242.666} C_DIS
LIN {X 0.138,Y -515.994,Z 778.143,A 0.000,B 0.000,C 90.000,E1 241.769} C_DIS
LIN {X 0.172,Y -513.772,Z 778.137,A 0.000,B 0.000,C 90.000,E1 240.589} C_DIS
LIN {X 0.075,Y -510.938,Z 778.129,A 0.000,B 0.000,C 90.000,E1 239.125} C_DIS
LIN {X 0.024,Y -508.640,Z 778.122,A 0.000,B 0.000,C 90.000,E1 237.946} C_DIS
LIN {X 0.048,Y -506.151,Z 778.115,A 0.000,B 0.000,C 90.000,E1 236.755} C_DIS
LIN {X -0.126,Y -504.243,Z 778.110,A 0.000,B 0.000,C 90.000,E1 235.881} C_DIS
LIN {X -0.157,Y -501.512,Z 778.104,A 0.000,B 0.000,C 90.000,E1 234.689} C_DIS
LIN {X -0.229,Y -498.579,Z 778.097,A 0.000,B 0.000,C 90.000,E1 233.497} C_DIS
LIN {X -0.018,Y -494.022,Z 778.087,A 0.000,B 0.000,C 90.000,E1 231.662} C_DIS
LIN {X -0.065,Y -490.301,Z 778.079,A 0.000,B 0.000,C 90.000,E1 230.150} C_DIS
LIN {X 0.041,Y -485.356,Z 778.067,A 0.000,B 0.000,C 90.000,E1 228.000} C_DIS
LIN {X 0.085,Y -482.018,Z 778.058,A 0.000,B 0.000,C 90.000,E1 226.458} C_DIS
LIN {X 0.013,Y -480.785,Z 778.055,A 0.000,B 0.000,C 90.000,E1 225.850} C_DIS
LIN {X -0.274,Y -476.706,Z 778.044,A 0.000,B 0.000,C 90.000,E1 224.028} C_DIS
LIN {X -0.069,Y -473.338,Z 778.036,A 0.000,B 0.000,C 90.000,E1 222.447} C_DIS
LIN {X 0.020,Y -467.878,Z 778.022,A 0.000,B 0.000,C 90.000,E1 219.930} C_DIS
LIN {X -0.212,Y -464.589,Z 778.013,A 0.000,B 0.000,C 90.000,E1 218.382} C_DIS
LIN {X -0.024,Y -460.627,Z 778.003,A 0.000,B 0.000,C 90.000,E1 216.457} C_DIS
LIN {X 0.070,Y -456.642,Z 777.992,A 0.000,B 0.000,C 90.000,E1 214.532} C_DIS
LIN {X -0.265,Y -451.505,Z 777.978,A 0.000,B 0.000,C 90.000,E1 212.005} C_DIS
LIN {X 0.166,Y -448.344,Z 777.969,A 0.000,B 0.000,C 90.000,E1 210.335} C_DIS
LIN {X -0.083,Y -445.277,Z 777.960,A 0.000,B 0.000,C 90.000,E1 208.743} C_DIS
LIN {X -0.215,Y -442.190,Z 777.951,A 0.000,B 0.000,C 90.000,E1 207.129} C_DIS
LIN {X -0.011,Y -439.049,Z 777.942,A 0.000,B 0.000,C 90.000,E1 205.463} C_DIS
LIN {X -0.062,Y -435.979,Z 777.932,A 0.000,B 0.000,C 90.000,E1 203.823} C_DIS
LIN {X 0.054,Y -432.847,Z 777.923,A 0.000,B 0.000,C 90.000,E1 202.153} C_DIS
LIN {X 0.106,Y -429.658,Z 777.914,A 0.000,B 0.000,C 90.000,E1 200.482} C_DIS
LIN {X 0.000,Y -425.841,Z 777.903,A 0.000,B 0.000,C 90.000,E1 198.489} C_DIS
LIN {X 0.029,Y -422.662,Z 777.893,A 0.000,B 0.000,C 90.000,E1 196.804} C_DIS
LIN {X 0.092,Y -417.988,Z 777.880,A 0.000,B 0.000,C 90.000,E1 194.426} C_DIS
LIN {X -0.126,Y -414.194,Z 777.869,A 0.000,B 0.000,C 90.000,E1 192.411} C_DIS
LIN {X 0.187,Y -410.458,Z 777.857,A 0.000,B 0.000,C 90.000,E1 190.310} C_DIS
LIN {X -0.109,Y -406.326,Z 777.844,A 0.000,B 0.000,C 90.000,E1 187.936} C_DIS
LIN {X -0.115,Y -403.434,Z 777.834,A 0.000,B 0.000,C 90.000,E1 186.201} C_DIS
LIN {X 0.018,Y -398.362,Z 777.817,A 0.000,B 0.000,C 90.000,E1 183.037} C_DIS
LIN {X 0.147,Y -393.399,Z 777.795,A 0.000,B 0.000,C 90.000,E1 179.141} C_DIS
LIN {X -0.053,Y -390.332,Z 777.780,A 0.000,B 0.000,C 90.000,E1 176.331} C_DIS
LIN {X -0.033,Y -388.661,Z 777.770,A 0.000,B 0.000,C 90.000,E1 174.546} C_DIS
LIN {X 0.207,Y -386.401,Z 777.756,A 0.000,B 0.000,C 90.000,E1 172.008} C_DIS
LIN {X -0.194,Y -384.941,Z 777.746,A 0.000,B 0.000,C 90.000,E1 170.274} C_DIS
LIN {X 0.173,Y -383.216,Z 777.732,A 0.000,B 0.000,C 90.000,E1 167.701} C_DIS
LIN {X 0.105,Y -381.476,Z 777.714,A 0.000,B 0.000,C 90.000,E1 164.464} C_DIS
LIN {X 0.009,Y -380.671,Z 777.704,A 0.000,B 0.000,C 90.000,E1 162.670} C_DIS
LIN {X 0.013,Y -379.906,Z 777.690,A 0.000,B 0.000,C 90.000,E1 160.134} C_DIS
LIN {X 0.063,Y -379.659,Z 777.661,A 0.000,B 0.000,C 90.000,E1 155.049} C_DIS
LIN {X 0.138,Y -381.147,Z 777.639,A 0.000,B 0.000,C 90.000,E1 151.051} C_DIS
LIN {X 0.047,Y -383.375,Z 777.625,A 0.000,B 0.000,C 90.000,E1 148.535} C_DIS
LIN {X 0.048,Y -384.755,Z 777.619,A 0.000,B 0.000,C 90.000,E1 147.454} C_DIS
LIN {X -0.008,Y -388.267,Z 777.607,A 0.000,B 0.000,C 90.000,E1 145.308} C_DIS
LIN {X -0.114,Y -389.806,Z 777.603,A 0.000,B 0.000,C 90.000,E1 144.609} C_DIS
LIN {X -0.209,Y -391.652,Z 777.599,A 0.000,B 0.000,C 90.000,E1 143.909} C_DIS
LIN {X -0.096,Y -394.464,Z 777.594,A 0.000,B 0.000,C 90.000,E1 143.004} C_DIS
LIN {X 0.084,Y -397.224,Z 777.591,A 0.000,B 0.000,C 90.000,E1 142.271} C_DIS
LIN {X 0.079,Y -399.731,Z 777.588,A 0.000,B 0.000,C 90.000,E1 141.743} C_DIS
LIN {X 0.073,Y -402.371,Z 777.585,A 0.000,B 0.000,C 90.000,E1 141.295} C_DIS
LIN {X 0.189,Y -406.744,Z 777.582,A 0.000,B 0.000,C 90.000,E1 140.642} C_DIS
LIN {X -0.113,Y -423.596,Z 777.570,A 0.000,B 0.000,C 90.000,E1 138.690} C_DIS
LIN {X 0.013,Y -440.733,Z 777.560,A 0.000,B 0.000,C 90.000,E1 136.824} C_DIS
LIN {X 0.189,Y -449.137,Z 777.555,A 0.000,B 0.000,C 90.000,E1 135.891} C_DIS
LIN {X -0.037,Y -458.646,Z 777.549,A 0.000,B 0.000,C 90.000,E1 134.838} C_DIS
LIN {X 0.151,Y -465.049,Z 777.545,A 0.000,B 0.000,C 90.000,E1 134.028} C_DIS
LIN {X 0.093,Y -472.563,Z 777.540,A 0.000,B 0.000,C 90.000,E1 133.095} C_DIS
LIN {X 0.124,Y -479.790,Z 777.534,A 0.000,B 0.000,C 90.000,E1 132.162} C_DIS
LIN {X 0.106,Y -485.525,Z 777.530,A 0.000,B 0.000,C 90.000,E1 131.391} C_DIS
LIN {X -0.160,Y -489.756,Z 777.527,A 0.000,B 0.000,C 90.000,E1 130.825} C_DIS
LIN {X 0.054,Y -495.982,Z 777.522,A 0.000,B 0.000,C 90.000,E1 129.886} C_DIS
LIN {X 0.186,Y -500.917,Z 777.517,A 0.000,B 0.000,C 90.000,E1 129.116} C_DIS
LIN {X 0.039,Y -508.111,Z 777.511,A 0.000,B 0.000,C 90.000,E1 127.935} C_DIS
LIN {X -0.044,Y -512.331,Z 777.507,A 0.000,B 0.000,C 90.000,E1 127.202} C_DIS
LIN {X 0.068,Y -518.696,Z 777.500,A 0.000,B 0.000,C 90.000,E1 126.011} C_DIS
LIN {X -0.275,Y -523.919,Z 777.494,A 0.000,B 0.000,C 90.000,E1 125.025} C_DIS
LIN {X 0.242,Y -526.046,Z 777.492,A 0.000,B 0.000,C 90.000,E1 124.532} C_DIS
LIN {X -0.091,Y -527.257,Z 777.490,A 0.000,B 0.000,C 90.000,E1 124.278} C_DIS
LIN {X 0.167,Y -529.769,Z 777.487,A 0.000,B 0.000,C 90.000,E1 123.706} C_DIS
LIN {X -0.187,Y -533.440,Z 777.483,A 0.000,B 0.000,C 90.000,E1 122.880} C_DIS
LIN {X -0.066,Y -538.087,Z 777.476,A 0.000,B 0.000,C 90.000,E1 121.720} C_DIS
LIN {X -0.167,Y -541.287,Z 777.471,A 0.000,B 0.000,C 90.000,E1 120.875} C_DIS
LIN {X -0.211,Y -545.211,Z 777.465,A 0.000,B 0.000,C 90.000,E1 119.745} C_DIS
LIN {X -0.204,Y -548.925,Z 777.459,A 0.000,B 0.000,C 90.000,E1 118.615} C_DIS
LIN {X 0.076,Y -552.382,Z 777.453,A 0.000,B 0.000,C 90.000,E1 117.462} C_DIS
LIN {X 0.141,Y -554.606,Z 777.448,A 0.000,B 0.000,C 90.000,E1 116.616} C_DIS
LIN {X -0.302,Y -555.867,Z 777.445,A 0.000,B 0.000,C 90.000,E1 116.104} C_DIS
LIN {X 0.293,Y -557.519,Z 777.440,A 0.000,B 0.000,C 90.000,E1 115.207} C_DIS
LIN {X -0.133,Y -558.499,Z 777.437,A 0.000,B 0.000,C 90.000,E1 114.695} C_DIS
LIN {X 0.255,Y -559.681,Z 777.433,A 0.000,B 0.000,C 90.000,E1 113.823} C_DIS
LIN {X 0.137,Y -561.991,Z 777.422,A 0.000,B 0.000,C 90.000,E1 111.897} C_DIS
LIN {X 0.154,Y -563.180,Z 777.416,A 0.000,B 0.000,C 90.000,E1 110.791} C_DIS
LIN {X -0.214,Y -564.530,Z 777.408,A 0.000,B 0.000,C 90.000,E1 109.450} C_DIS
LIN {X -0.028,Y -565.712,Z 777.400,A 0.000,B 0.000,C 90.000,E1 108.055} C_DIS
LIN {X 0.165,Y -566.983,Z 777.391,A 0.000,B 0.000,C 90.000,E1 106.386} C_DIS
LIN {X 0.220,Y -568.060,Z 777.384,A 0.000,B 0.000,C 90.000,E1 105.009} C_DIS
LIN {X -0.054,Y -569.620,Z 777.373,A 0.000,B 0.000,C 90.000,E1 103.119} C_DIS
LIN {X 0.140,Y -571.313,Z 777.362,A 0.000,B 0.000,C 90.000,E1 101.186} C_DIS
LIN {X 0.071,Y -572.688,Z 777.353,A 0.000,B 0.000,C 90.000,E1 99.557} C_DIS
LIN {X 0.198,Y -573.590,Z 777.347,A 0.000,B 0.000,C 90.000,E1 98.454} C_DIS
LIN {X -0.112,Y -574.659,Z 777.340,A 0.000,B 0.000,C 90.000,E1 97.125} C_DIS
LIN {X 0.166,Y -575.577,Z 777.332,A 0.000,B 0.000,C 90.000,E1 95.739} C_DIS
LIN {X -0.030,Y -576.587,Z 777.323,A 0.000,B 0.000,C 90.000,E1 94.131} C_DIS
LIN {X 0.219,Y -577.371,Z 777.315,A 0.000,B 0.000,C 90.000,E1 92.751} C_DIS
LIN {X 0.286,Y -577.945,Z 777.309,A 0.000,B 0.000,C 90.000,E1 91.661} C_DIS
LIN {X 0.091,Y -578.684,Z 777.300,A 0.000,B 0.000,C 90.000,E1 90.057} C_DIS
LIN {X 0.164,Y -579.110,Z 777.294,A 0.000,B 0.000,C 90.000,E1 88.969} C_DIS
LIN {X 0.006,Y -579.656,Z 777.285,A 0.000,B 0.000,C 90.000,E1 87.364} C_DIS
LIN {X -0.108,Y -580.092,Z 777.276,A 0.000,B 0.000,C 90.000,E1 85.755} C_DIS
LIN {X -0.217,Y -580.436,Z 777.267,A 0.000,B 0.000,C 90.000,E1 84.147} C_DIS
LIN {X -0.051,Y -580.697,Z 777.257,A 0.000,B 0.000,C 90.000,E1 82.243} C_DIS
LIN {X -0.161,Y -580.825,Z 777.249,A 0.000,B 0.000,C 90.000,E1 80.905} C_DIS
LIN {X 0.312,Y -580.905,Z 777.242,A 0.000,B 0.000,C 90.000,E1 79.511} C_DIS
LIN {X 0.204,Y -580.838,Z 777.234,A 0.000,B 0.000,C 90.000,E1 78.173} C_DIS
LIN {X 0.207,Y -580.712,Z 777.227,A 0.000,B 0.000,C 90.000,E1 76.825} C_DIS
LIN {X 0.002,Y -580.306,Z 777.218,A 0.000,B 0.000,C 90.000,E1 75.227} C_DIS
LIN {X 0.128,Y -579.876,Z 777.211,A 0.000,B 0.000,C 90.000,E1 73.866} C_DIS
LIN {X -0.150,Y -579.458,Z 777.203,A 0.000,B 0.000,C 90.000,E1 72.543} C_DIS
LIN {X -0.049,Y -578.756,Z 777.194,A 0.000,B 0.000,C 90.000,E1 70.913} C_DIS
LIN {X -0.155,Y -578.082,Z 777.186,A 0.000,B 0.000,C 90.000,E1 69.571} C_DIS
LIN {X 0.103,Y -577.093,Z 777.177,A 0.000,B 0.000,C 90.000,E1 67.922} C_DIS
LIN {X 0.167,Y -576.072,Z 777.170,A 0.000,B 0.000,C 90.000,E1 66.561} C_DIS
LIN {X -0.081,Y -574.952,Z 777.162,A 0.000,B 0.000,C 90.000,E1 65.229} C_DIS
LIN {X -0.183,Y -573.905,Z 777.156,A 0.000,B 0.000,C 90.000,E1 64.152} C_DIS
LIN {X -0.045,Y -572.658,Z 777.150,A 0.000,B 0.000,C 90.000,E1 63.050} C_DIS
LIN {X -0.187,Y -571.217,Z 777.144,A 0.000,B 0.000,C 90.000,E1 61.975} C_DIS
LIN {X 0.186,Y -569.585,Z 777.138,A 0.000,B 0.000,C 90.000,E1 60.845} C_DIS
LIN {X -0.234,Y -567.659,Z 777.132,A 0.000,B 0.000,C 90.000,E1 59.793} C_DIS
LIN {X -0.010,Y -566.067,Z 777.128,A 0.000,B 0.000,C 90.000,E1 58.948} C_DIS
LIN {X 0.003,Y -564.268,Z 777.123,A 0.000,B 0.000,C 90.000,E1 58.122} C_DIS
LIN {X -0.202,Y -561.604,Z 777.117,A 0.000,B 0.000,C 90.000,E1 57.041} C_DIS
LIN {X -0.137,Y -558.477,Z 777.111,A 0.000,B 0.000,C 90.000,E1 55.928} C_DIS
LIN {X -0.278,Y -556.854,Z 777.108,A 0.000,B 0.000,C 90.000,E1 55.388} C_DIS
LIN {X -0.036,Y -554.135,Z 777.103,A 0.000,B 0.000,C 90.000,E1 54.529} C_DIS
LIN {X -0.145,Y -551.127,Z 777.098,A 0.000,B 0.000,C 90.000,E1 53.703} C_DIS
LIN {X -0.021,Y -548.950,Z 777.095,A 0.000,B 0.000,C 90.000,E1 53.130} C_DIS
LIN {X 0.134,Y -545.307,Z 777.091,A 0.000,B 0.000,C 90.000,E1 52.271} C_DIS
LIN {X -0.033,Y -541.967,Z 777.087,A 0.000,B 0.000,C 90.000,E1 51.582} C_DIS
LIN {X 0.020,Y -539.149,Z 777.083,A 0.000,B 0.000,C 90.000,E1 51.009} C_DIS
LIN {X 0.048,Y -536.064,Z 777.080,A 0.000,B 0.000,C 90.000,E1 50.436} C_DIS
LIN {X -0.190,Y -531.720,Z 777.076,A 0.000,B 0.000,C 90.000,E1 49.747} C_DIS
LIN {X 0.125,Y -527.907,Z 777.073,A 0.000,B 0.000,C 90.000,E1 49.138} C_DIS
LIN {X 0.061,Y -523.562,Z 777.070,A 0.000,B 0.000,C 90.000,E1 48.566} C_DIS
LIN {X -0.227,Y -520.015,Z 777.068,A 0.000,B 0.000,C 90.000,E1 48.162} C_DIS
LIN {X 0.019,Y -514.822,Z 777.064,A 0.000,B 0.000,C 90.000,E1 47.553} C_DIS
LIN {X 0.159,Y -509.474,Z 777.061,A 0.000,B 0.000,C 90.000,E1 46.986} C_DIS
LIN {X -0.224,Y -505.276,Z 777.059,A 0.000,B 0.000,C 90.000,E1 46.620} C_DIS
LIN {X 0.118,Y -499.232,Z 777.056,A 0.000,B 0.000,C 90.000,E1 46.053} C_DIS
LIN {X 0.020,Y -493.115,Z 777.053,A 0.000,B 0.000,C 90.000,E1 45.567} C_DIS
LIN {X 0.068,Y -488.532,Z 777.051,A 0.000,B 0.000,C 90.000,E1 45.202} C_DIS
LIN {X -0.047,Y -480.548,Z 777.048,A 0.000,B 0.000,C 90.000,E1 44.636} C_DIS
LIN {X 0.177,Y -470.908,Z 777.044,A 0.000,B 0.000,C 90.000,E1 43.947} C_DIS
LIN {X 0.076,Y -462.793,Z 777.041,A 0.000,B 0.000,C 90.000,E1 43.419} C_DIS
LIN {X 0.048,Y -448.333,Z 777.036,A 0.000,B 0.000,C 90.000,E1 42.447} C_DIS
LIN {X -0.218,Y -429.328,Z 777.029,A 0.000,B 0.000,C 90.000,E1 41.148} C_DIS
LIN {X -0.162,Y -416.674,Z 777.023,A 0.000,B 0.000,C 90.000,E1 40.172} C_DIS
LIN {X -0.075,Y -410.547,Z 777.020,A 0.000,B 0.000,C 90.000,E1 39.644} C_DIS
LIN {X 0.209,Y -407.218,Z 777.018,A 0.000,B 0.000,C 90.000,E1 39.277} C_DIS
LIN {X 0.177,Y -407.192,Z 777.018,A 0.000,B 0.000,C 90.000,E1 39.277} C_DIS
LIN {X -0.197,Y -405.757,Z 777.014,A 0.000,B 0.000,C 90.000,E1 38.463} C_DIS
LIN {X 0.120,Y -397.761,Z 776.991,A 0.000,B 0.000,C 90.000,E1 34.405} C_DIS
LIN {X 0.007,Y -397.563,Z 776.990,A 0.000,B 0.000,C 90.000,E1 34.246} C_DIS
LIN {X -0.034,Y -398.272,Z 776.974,A 0.000,B 0.000,C 90.000,E1 31.258} C_DIS
LIN {X 0.049,Y -399.478,Z 776.958,A 0.000,B 0.000,C 90.000,E1 28.437} C_DIS
LIN {X 0.101,Y -400.851,Z 776.944,A 0.000,B 0.000,C 90.000,E1 25.976} C_DIS
LIN {X -0.131,Y -403.246,Z 776.925,A 0.000,B 0.000,C 90.000,E1 22.514} C_DIS
LIN {X -0.011,Y -406.915,Z 776.904,A 0.000,B 0.000,C 90.000,E1 18.671} C_DIS
LIN {X 0.166,Y -411.430,Z 776.885,A 0.000,B 0.000,C 90.000,E1 15.190} C_DIS
LIN {X -0.085,Y -415.636,Z 776.869,A 0.000,B 0.000,C 90.000,E1 12.479} C_DIS
LIN {X -0.014,Y -419.090,Z 776.858,A 0.000,B 0.000,C 90.000,E1 10.423} C_DIS
LIN {X -0.088,Y -422.596,Z 776.847,A 0.000,B 0.000,C 90.000,E1 8.398} C_DIS
LIN {X -0.160,Y -425.489,Z 776.837,A 0.000,B 0.000,C 90.000,E1 6.720} C_DIS
LIN {X 0.020,Y -430.288,Z 776.822,A 0.000,B 0.000,C 90.000,E1 4.012} C_DIS
LIN {X -0.174,Y -435.359,Z 776.808,A 0.000,B 0.000,C 90.000,E1 1.375} C_DIS
LIN {X -0.055,Y -439.754,Z 776.795,A 0.000,B 0.000,C 90.000,E1 359.141} C_DIS
LIN {X -0.066,Y -444.692,Z 776.782,A 0.000,B 0.000,C 90.000,E1 356.846} C_DIS
LIN {X 0.099,Y -449.989,Z 776.770,A 0.000,B 0.000,C 90.000,E1 354.546} C_DIS
LIN {X 0.084,Y -453.778,Z 776.761,A 0.000,B 0.000,C 90.000,E1 352.932} C_DIS
LIN {X 0.132,Y -457.533,Z 776.752,A 0.000,B 0.000,C 90.000,E1 351.319} C_DIS
LIN {X 0.147,Y -460.422,Z 776.745,A 0.000,B 0.000,C 90.000,E1 350.038} C_DIS
LIN {X 0.209,Y -463.193,Z 776.738,A 0.000,B 0.000,C 90.000,E1 348.757} C_DIS
LIN {X -0.046,Y -466.084,Z 776.731,A 0.000,B 0.000,C 90.000,E1 347.521} C_DIS
LIN {X 0.020,Y -467.846,Z 776.727,A 0.000,B 0.000,C 90.000,E1 346.881} C_DIS
LIN {X -0.173,Y -468.831,Z 776.725,A 0.000,B 0.000,C 90.000,E1 346.589} C_DIS
LIN {X -0.167,Y -470.697,Z 776.723,A 0.000,B 0.000,C 90.000,E1 346.117} C_DIS
LIN {X -0.153,Y -473.240,Z 776.720,A 0.000,B 0.000,C 90.000,E1 345.644} C_DIS
LIN {X 0.228,Y -475.755,Z 776.718,A 0.000,B 0.000,C 90.000,E1 345.227} C_DIS
LIN {X -0.142,Y -479.966,Z 776.716,A 0.000,B 0.000,C 90.000,E1 344.810} C_DIS
LIN {X -0.098,Y -485.517,Z 776.713,A 0.000,B 0.000,C 90.000,E1 344.283} C_DIS
LIN {X -0.112,Y -494.227,Z 776.709,A 0.000,B 0.000,C 90.000,E1 343.614} C_DIS
LIN {X 0.241,Y -514.428,Z 776.701,A 0.000,B 0.000,C 90.000,E1 342.181} C_DIS
LIN {X -0.308,Y -530.163,Z 776.696,A 0.000,B 0.000,C 90.000,E1 341.221} C_DIS
LIN {X 0.016,Y -536.342,Z 776.693,A 0.000,B 0.000,C 90.000,E1 340.786} C_DIS
LIN {X -0.186,Y -545.690,Z 776.690,A 0.000,B 0.000,C 90.000,E1 340.188} C_DIS
LIN {X -0.203,Y -551.425,Z 776.687,A 0.000,B 0.000,C 90.000,E1 339.752} C_DIS
LIN {X 0.043,Y -558.351,Z 776.684,A 0.000,B 0.000,C 90.000,E1 339.135} C_DIS
LIN {X 0.078,Y -563.447,Z 776.681,A 0.000,B 0.000,C 90.000,E1 338.646} C_DIS
LIN {X 0.202,Y -569.655,Z 776.678,A 0.000,B 0.000,C 90.000,E1 337.975} C_DIS
LIN {X -0.335,Y -574.489,Z 776.675,A 0.000,B 0.000,C 90.000,E1 337.486} C_DIS
LIN {X -0.053,Y -577.932,Z 776.673,A 0.000,B 0.000,C 90.000,E1 337.050} C_DIS
LIN {X -0.023,Y -585.221,Z 776.667,A 0.000,B 0.000,C 90.000,E1 336.102} C_DIS
LIN {X 0.156,Y -591.186,Z 776.663,A 0.000,B 0.000,C 90.000,E1 335.281} C_DIS
LIN {X 0.143,Y -596.823,Z 776.658,A 0.000,B 0.000,C 90.000,E1 334.485} C_DIS
LIN {X 0.097,Y -603.886,Z 776.653,A 0.000,B 0.000,C 90.000,E1 333.435} C_DIS
LIN {X -0.094,Y -609.672,Z 776.647,A 0.000,B 0.000,C 90.000,E1 332.538} C_DIS
LIN {X -0.251,Y -616.820,Z 776.641,A 0.000,B 0.000,C 90.000,E1 331.385} C_DIS
LIN {X 0.004,Y -620.590,Z 776.637,A 0.000,B 0.000,C 90.000,E1 330.717} C_DIS
LIN {X 0.309,Y -627.199,Z 776.631,A 0.000,B 0.000,C 90.000,E1 329.537} C_DIS
LIN {X 0.133,Y -631.342,Z 776.627,A 0.000,B 0.000,C 90.000,E1 328.791} C_DIS
LIN {X 0.016,Y -635.832,Z 776.622,A 0.000,B 0.000,C 90.000,E1 327.916} C_DIS
LIN {X -0.035,Y -640.653,Z 776.616,A 0.000,B 0.000,C 90.000,E1 326.914} C_DIS
LIN {X 0.322,Y -645.224,Z 776.611,A 0.000,B 0.000,C 90.000,E1 325.881} C_DIS
LIN {X 0.207,Y -649.497,Z 776.605,A 0.000,B 0.000,C 90.000,E1 324.895} C_DIS
LIN {X 0.151,Y -653.471,Z 776.600,A 0.000,B 0.000,C 90.000,E1 323.909} C_DIS
LIN {X 0.141,Y -657.132,Z 776.594,A 0.000,B 0.000,C 90.000,E1 322.924} C_DIS
LIN {X -0.351,Y -660.615,Z 776.589,A 0.000,B 0.000,C 90.000,E1 321.984} C_DIS
LIN {X 0.128,Y -663.934,Z 776.583,A 0.000,B 0.000,C 90.000,E1 320.964} C_DIS
LIN {X 0.129,Y -667.770,Z 776.576,A 0.000,B 0.000,C 90.000,E1 319.747} C_DIS
LIN {X 0.193,Y -670.692,Z 776.571,A 0.000,B 0.000,C 90.000,E1 318.771} C_DIS
LIN {X 0.307,Y -674.070,Z 776.564,A 0.000,B 0.000,C 90.000,E1 317.553} C_DIS
LIN {X 0.004,Y -677.418,Z 776.556,A 0.000,B 0.000,C 90.000,E1 316.134} C_DIS
LIN {X 0.194,Y -679.940,Z 776.550,A 0.000,B 0.000,C 90.000,E1 314.919} C_DIS
LIN {X 0.329,Y -681.333,Z 776.546,A 0.000,B 0.000,C 90.000,E1 314.190} C_DIS
LIN {X 0.163,Y -683.893,Z 776.538,A 0.000,B 0.000,C 90.000,E1 312.771} C_DIS
LIN {X -0.078,Y -685.490,Z 776.532,A 0.000,B 0.000,C 90.000,E1 311.838} C_DIS
LIN {X 0.275,Y -687.177,Z 776.526,A 0.000,B 0.000,C 90.000,E1 310.620} C_DIS
LIN {X -0.377,Y -688.374,Z 776.521,A 0.000,B 0.000,C 90.000,E1 309.725} C_DIS
LIN {X 0.175,Y -689.965,Z 776.513,A 0.000,B 0.000,C 90.000,E1 308.257} C_DIS
LIN {X 0.150,Y -691.125,Z 776.506,A 0.000,B 0.000,C 90.000,E1 307.076} C_DIS
LIN {X -0.080,Y -692.396,Z 776.498,A 0.000,B 0.000,C 90.000,E1 305.678} C_DIS
LIN {X 0.076,Y -693.328,Z 776.492,A 0.000,B 0.000,C 90.000,E1 304.485} C_DIS
LIN {X 0.119,Y -694.551,Z 776.482,A 0.000,B 0.000,C 90.000,E1 302.832} C_DIS
LIN {X -0.188,Y -695.906,Z 776.473,A 0.000,B 0.000,C 90.000,E1 301.209} C_DIS
LIN {X 0.219,Y -696.676,Z 776.467,A 0.000,B 0.000,C 90.000,E1 300.001} C_DIS
LIN {X -0.066,Y -697.290,Z 776.459,A 0.000,B 0.000,C 90.000,E1 298.615} C_DIS
LIN {X -0.148,Y -698.118,Z 776.449,A 0.000,B 0.000,C 90.000,E1 296.744} C_DIS
LIN {X 0.118,Y -699.261,Z 776.438,A 0.000,B 0.000,C 90.000,E1 294.847} C_DIS
LIN {X 0.015,Y -699.222,Z 776.436,A 0.000,B 0.000,C 90.000,E1 294.387} C_DIS
LIN {X -0.005,Y -699.149,Z 776.434,A 0.000,B 0.000,C 90.000,E1 294.155} C_DIS
LIN {X 0.261,Y -698.687,Z 776.433,A 0.000,B 0.000,C 90.000,E1 293.898} C_DIS
LIN {X -0.130,Y -697.307,Z 776.430,A 0.000,B 0.000,C 90.000,E1 293.462} C_DIS
LIN {X 0.000,Y -696.706,Z 776.430,A 0.000,B 0.000,C 90.000,E1 293.334} C_DIS
LIN {X 0.256,Y -694.720,Z 776.428,A 0.000,B 0.000,C 90.000,E1 293.078} C_DIS
LIN {X -0.246,Y -691.089,Z 776.426,A 0.000,B 0.000,C 90.000,E1 292.770} C_DIS
LIN {X -0.095,Y -689.418,Z 776.426,A 0.000,B 0.000,C 90.000,E1 292.642} C_DIS
LIN {X -0.109,Y -683.167,Z 776.424,A 0.000,B 0.000,C 90.000,E1 292.386} C_DIS
LIN {X -0.126,Y -676.761,Z 776.423,A 0.000,B 0.000,C 90.000,E1 292.206} C_DIS
LIN {X -0.109,Y -674.662,Z 776.423,A 0.000,B 0.000,C 90.000,E1 292.153} C_DIS
LIN {X -0.009,Y -663.729,Z 776.422,A 0.000,B 0.000,C 90.000,E1 291.972} C_DIS
LIN {X 0.007,Y -655.018,Z 776.421,A 0.000,B 0.000,C 90.000,E1 291.844} C_DIS
LIN {X 0.087,Y -644.780,Z 776.420,A 0.000,B 0.000,C 90.000,E1 291.663} C_DIS
LIN {X -0.155,Y -631.187,Z 776.419,A 0.000,B 0.000,C 90.000,E1 291.408} C_DIS
LIN {X 0.267,Y -614.106,Z 776.417,A 0.000,B 0.000,C 90.000,E1 290.972} C_DIS
LIN {X 0.284,Y -593.287,Z 776.414,A 0.000,B 0.000,C 90.000,E1 290.429} C_DIS
LIN {X -0.068,Y -567.522,Z 776.409,A 0.000,B 0.000,C 90.000,E1 289.685} C_DIS
LIN {X 0.153,Y -563.957,Z 776.409,A 0.000,B 0.000,C 90.000,E1 289.523} C_DIS
LIN {X 0.166,Y -559.925,Z 776.408,A 0.000,B 0.000,C 90.000,E1 289.341} C_DIS
LIN {X -0.098,Y -557.307,Z 776.406,A 0.000,B 0.000,C 90.000,E1 289.141} C_DIS
LIN {X -0.207,Y -556.701,Z 776.406,A 0.000,B 0.000,C 90.000,E1 289.033} C_DIS
LIN {X 0.203,Y -556.131,Z 776.405,A 0.000,B 0.000,C 90.000,E1 288.852} C_DIS
LIN {X -0.059,Y -555.580,Z 776.403,A 0.000,B 0.000,C 90.000,E1 288.598} C_DIS
LIN {X 0.052,Y -555.184,Z 776.402,A 0.000,B 0.000,C 90.000,E1 288.308} C_DIS
LIN {X 0.202,Y -554.724,Z 776.397,A 0.000,B 0.000,C 90.000,E1 287.457} C_DIS
LIN {X 0.062,Y -554.486,Z 776.394,A 0.000,B 0.000,C 90.000,E1 286.913} C_DIS
LIN {X -0.295,Y -553.404,Z 776.382,A 0.000,B 0.000,C 90.000,E1 284.717} C_DIS
LIN {X 0.026,Y -552.808,Z 776.372,A 0.000,B 0.000,C 90.000,E1 283.008} C_DIS
LIN {X 0.324,Y -552.234,Z 776.363,A 0.000,B 0.000,C 90.000,E1 281.299} C_DIS
LIN {X -0.043,Y -551.621,Z 776.352,A 0.000,B 0.000,C 90.000,E1 279.378} C_DIS
LIN {X 0.033,Y -551.080,Z 776.341,A 0.000,B 0.000,C 90.000,E1 277.409} C_DIS
LIN {X 0.219,Y -550.750,Z 776.337,A 0.000,B 0.000,C 90.000,E1 276.549} C_DIS
LIN {X -0.034,Y -550.140,Z 776.330,A 0.000,B 0.000,C 90.000,E1 275.454} C_DIS
LIN {X -0.119,Y -548.796,Z 776.319,A 0.000,B 0.000,C 90.000,E1 273.498} C_DIS
LIN {X 0.262,Y -547.642,Z 776.308,A 0.000,B 0.000,C 90.000,E1 271.489} C_DIS
LIN {X -0.054,Y -546.728,Z 776.301,A 0.000,B 0.000,C 90.000,E1 270.115} C_DIS
LIN {X 0.161,Y -545.784,Z 776.293,A 0.000,B 0.000,C 90.000,E1 268.682} C_DIS
LIN {X -0.079,Y -544.479,Z 776.282,A 0.000,B 0.000,C 90.000,E1 266.731} C_DIS
LIN {X 0.192,Y -543.271,Z 776.271,A 0.000,B 0.000,C 90.000,E1 264.723} C_DIS
LIN {X -0.098,Y -542.308,Z 776.263,A 0.000,B 0.000,C 90.000,E1 263.337} C_DIS
LIN {X 0.062,Y -541.322,Z 776.257,A 0.000,B 0.000,C 90.000,E1 262.186} C_DIS
LIN {X -0.038,Y -539.719,Z 776.246,A 0.000,B 0.000,C 90.000,E1 260.208} C_DIS
LIN {X -0.174,Y -537.938,Z 776.235,A 0.000,B 0.000,C 90.000,E1 258.229} C_DIS
LIN {X 0.140,Y -536.650,Z 776.227,A 0.000,B 0.000,C 90.000,E1 256.769} C_DIS
LIN {X -0.083,Y -535.842,Z 776.222,A 0.000,B 0.000,C 90.000,E1 255.936} C_DIS
LIN {X 0.024,Y -533.639,Z 776.211,A 0.000,B 0.000,C 90.000,E1 253.921} C_DIS
LIN {X 0.184,Y -531.669,Z 776.201,A 0.000,B 0.000,C 90.000,E1 252.181} C_DIS
LIN {X 0.097,Y -530.366,Z 776.195,A 0.000,B 0.000,C 90.000,E1 251.040} C_DIS
LIN {X -0.151,Y -528.356,Z 776.187,A 0.000,B 0.000,C 90.000,E1 249.625} C_DIS
LIN {X 0.241,Y -525.907,Z 776.177,A 0.000,B 0.000,C 90.000,E1 247.847} C_DIS
LIN {X -0.034,Y -522.791,Z 776.166,A 0.000,B 0.000,C 90.000,E1 245.845} C_DIS
LIN {X -0.040,Y -521.399,Z 776.161,A 0.000,B 0.000,C 90.000,E1 244.973} C_DIS
LIN {X 0.107,Y -518.523,Z 776.151,A 0.000,B 0.000,C 90.000,E1 243.204} C_DIS
LIN {X 0.173,Y -516.531,Z 776.145,A 0.000,B 0.000,C 90.000,E1 242.025} C_DIS
LIN {X -0.035,Y -514.348,Z 776.138,A 0.000,B 0.000,C 90.000,E1 240.873} C_DIS
LIN {X 0.214,Y -510.908,Z 776.128,A 0.000,B 0.000,C 90.000,E1 239.076} C_DIS
LIN {X -0.005,Y -508.611,Z 776.122,A 0.000,B 0.000,C 90.000,E1 237.916} C_DIS
LIN {X 0.173,Y -506.104,Z 776.115,A 0.000,B 0.000,C 90.000,E1 236.707} C_DIS
LIN {X 0.276,Y -504.193,Z 776.110,A 0.000,B 0.000,C 90.000,E1 235.801} C_DIS
LIN {X -0.044,Y -501.456,Z 776.104,A 0.000,B 0.000,C 90.000,E1 234.642} C_DIS
LIN {X 0.174,Y -498.505,Z 776.097,A 0.000,B 0.000,C 90.000,E1 233.417} C_DIS
LIN {X 0.075,Y -493.934,Z 776.087,A 0.000,B 0.000,C 90.000,E1 231.618} C_DIS
LIN {X -0.204,Y -490.972,Z 776.080,A 0.000,B 0.000,C 90.000,E1 230.436} C_DIS
LIN {X 0.288,Y -486.018,Z 776.068,A 0.000,B 0.000,C 90.000,E1 228.243} C_DIS
LIN {X 0.057,Y -480.763,Z 776.055,A 0.000,B 0.000,C 90.000,E1 225.810} C_DIS
LIN {X 0.111,Y -476.676,Z 776.044,A 0.000,B 0.000,C 90.000,E1 223.947} C_DIS
LIN {X -0.008,Y -473.309,Z 776.036,A 0.000,B 0.000,C 90.000,E1 222.405} C_DIS
LIN {X 0.094,Y -467.843,Z 776.022,A 0.000,B 0.000,C 90.000,E1 219.886} C_DIS
LIN {X 0.156,Y -464.514,Z 776.013,A 0.000,B 0.000,C 90.000,E1 218.302} C_DIS
LIN {X -0.056,Y -461.264,Z 776.004,A 0.000,B 0.000,C 90.000,E1 216.744} C_DIS
LIN {X -0.055,Y -457.937,Z 775.995,A 0.000,B 0.000,C 90.000,E1 215.152} C_DIS
LIN {X 0.176,Y -453.341,Z 775.983,A 0.000,B 0.000,C 90.000,E1 212.880} C_DIS
LIN {X 0.167,Y -450.850,Z 775.976,A 0.000,B 0.000,C 90.000,E1 211.592} C_DIS
LIN {X -0.037,Y -445.904,Z 775.961,A 0.000,B 0.000,C 90.000,E1 209.027} C_DIS
LIN {X -0.096,Y -442.174,Z 775.950,A 0.000,B 0.000,C 90.000,E1 207.078} C_DIS
LIN {X 0.111,Y -439.032,Z 775.941,A 0.000,B 0.000,C 90.000,E1 205.412} C_DIS
LIN {X 0.064,Y -435.965,Z 775.932,A 0.000,B 0.000,C 90.000,E1 203.770} C_DIS
LIN {X -0.217,Y -432.828,Z 775.923,A 0.000,B 0.000,C 90.000,E1 202.153} C_DIS
LIN {X 0.051,Y -429.057,Z 775.912,A 0.000,B 0.000,C 90.000,E1 200.120} C_DIS
LIN {X -0.067,Y -425.211,Z 775.901,A 0.000,B 0.000,C 90.000,E1 198.127} C_DIS
LIN {X -0.235,Y -422.644,Z 775.893,A 0.000,B 0.000,C 90.000,E1 196.804} C_DIS
LIN {X -0.012,Y -417.353,Z 775.878,A 0.000,B 0.000,C 90.000,E1 194.064} C_DIS
LIN {X 0.064,Y -413.542,Z 775.867,A 0.000,B 0.000,C 90.000,E1 192.007} C_DIS
LIN {X -0.038,Y -409.903,Z 775.855,A 0.000,B 0.000,C 90.000,E1 189.962} C_DIS
LIN {X 0.055,Y -405.749,Z 775.842,A 0.000,B 0.000,C 90.000,E1 187.530} C_DIS
LIN {X 0.034,Y -403.468,Z 775.834,A 0.000,B 0.000,C 90.000,E1 186.144} C_DIS
LIN {X 0.116,Y -397.943,Z 775.815,A 0.000,B 0.000,C 90.000,E1 182.636} C_DIS
LIN {X -0.023,Y -393.907,Z 775.797,A 0.000,B 0.000,C 90.000,E1 179.484} C_DIS
LIN {X 0.100,Y -390.411,Z 775.779,A 0.000,B 0.000,C 90.000,E1 176.274} C_DIS
LIN {X 0.021,Y -388.449,Z 775.768,A 0.000,B 0.000,C 90.000,E1 174.147} C_DIS
LIN {X -0.021,Y -386.544,Z 775.756,A 0.000,B 0.000,C 90.000,E1 172.008} C_DIS
LIN {X -0.045,Y -384.863,Z 775.744,A 0.000,B 0.000,C 90.000,E1 169.859} C_DIS
LIN {X -0.044,Y -383.469,Z 775.732,A 0.000,B 0.000,C 90.000,E1 167.701} C_DIS
LIN {X 0.000,Y -381.757,Z 775.714,A 0.000,B 0.000,C 90.000,E1 164.448} C_DIS
LIN {X -0.186,Y -380.716,Z 775.700,A 0.000,B 0.000,C 90.000,E1 161.945} C_DIS
LIN {X -0.050,Y -380.108,Z 775.688,A 0.000,B 0.000,C 90.000,E1 159.752} C_DIS
LIN {X -0.112,Y -379.954,Z 775.661,A 0.000,B 0.000,C 90.000,E1 155.049} C_DIS
LIN {X -0.061,Y -381.853,Z 775.635,A 0.000,B 0.000,C 90.000,E1 150.333} C_DIS
LIN {X -0.111,Y -383.538,Z 775.625,A 0.000,B 0.000,C 90.000,E1 148.535} C_DIS
LIN {X -0.217,Y -387.540,Z 775.609,A 0.000,B 0.000,C 90.000,E1 145.674} C_DIS
LIN {X 0.046,Y -389.712,Z 775.603,A 0.000,B 0.000,C 90.000,E1 144.562} C_DIS
LIN {X -0.053,Y -391.444,Z 775.599,A 0.000,B 0.000,C 90.000,E1 143.863} C_DIS
LIN {X 0.095,Y -393.469,Z 775.595,A 0.000,B 0.000,C 90.000,E1 143.130} C_DIS
LIN {X 0.178,Y -394.765,Z 775.593,A 0.000,B 0.000,C 90.000,E1 142.763} C_DIS
LIN {X 0.027,Y -395.931,Z 775.591,A 0.000,B 0.000,C 90.000,E1 142.431} C_DIS
LIN {X -0.094,Y -399.049,Z 775.587,A 0.000,B 0.000,C 90.000,E1 141.743} C_DIS
LIN {X -0.188,Y -402.381,Z 775.584,A 0.000,B 0.000,C 90.000,E1 141.170} C_DIS
LIN {X 0.084,Y -406.520,Z 775.581,A 0.000,B 0.000,C 90.000,E1 140.517} C_DIS
LIN {X -0.035,Y -414.023,Z 775.576,A 0.000,B 0.000,C 90.000,E1 139.622} C_DIS
LIN {X 0.218,Y -435.448,Z 775.563,A 0.000,B 0.000,C 90.000,E1 137.229} C_DIS
LIN {X -0.218,Y -444.025,Z 775.558,A 0.000,B 0.000,C 90.000,E1 136.377} C_DIS
LIN {X 0.195,Y -450.964,Z 775.553,A 0.000,B 0.000,C 90.000,E1 135.567} C_DIS
LIN {X -0.042,Y -457.713,Z 775.549,A 0.000,B 0.000,C 90.000,E1 134.838} C_DIS
LIN {X -0.074,Y -463.805,Z 775.545,A 0.000,B 0.000,C 90.000,E1 134.109} C_DIS
LIN {X 0.130,Y -471.482,Z 775.540,A 0.000,B 0.000,C 90.000,E1 133.137} C_DIS
LIN {X 0.104,Y -479.843,Z 775.534,A 0.000,B 0.000,C 90.000,E1 132.081} C_DIS
LIN {X 0.142,Y -484.406,Z 775.531,A 0.000,B 0.000,C 90.000,E1 131.472} C_DIS
LIN {X 0.169,Y -489.883,Z 775.526,A 0.000,B 0.000,C 90.000,E1 130.701} C_DIS
LIN {X 0.247,Y -495.123,Z 775.522,A 0.000,B 0.000,C 90.000,E1 129.930} C_DIS
LIN {X 0.144,Y -501.083,Z 775.517,A 0.000,B 0.000,C 90.000,E1 129.036} C_DIS
LIN {X -0.108,Y -507.447,Z 775.511,A 0.000,B 0.000,C 90.000,E1 128.016} C_DIS
LIN {X 0.014,Y -512.544,Z 775.506,A 0.000,B 0.000,C 90.000,E1 127.111} C_DIS
LIN {X 0.028,Y -518.946,Z 775.500,A 0.000,B 0.000,C 90.000,E1 125.931} C_DIS
LIN {X 0.317,Y -523.425,Z 775.495,A 0.000,B 0.000,C 90.000,E1 125.025} C_DIS
LIN {X 0.103,Y -525.614,Z 775.492,A 0.000,B 0.000,C 90.000,E1 124.612} C_DIS
LIN {X -0.101,Y -527.509,Z 775.490,A 0.000,B 0.000,C 90.000,E1 124.199} C_DIS
LIN {X 0.005,Y -529.382,Z 775.488,A 0.000,B 0.000,C 90.000,E1 123.785} C_DIS
LIN {X 0.094,Y -533.075,Z 775.483,A 0.000,B 0.000,C 90.000,E1 122.911} C_DIS
LIN {X -0.078,Y -536.027,Z 775.479,A 0.000,B 0.000,C 90.000,E1 122.212} C_DIS
LIN {X 0.081,Y -539.372,Z 775.474,A 0.000,B 0.000,C 90.000,E1 121.337} C_DIS
LIN {X 0.009,Y -543.504,Z 775.468,A 0.000,B 0.000,C 90.000,E1 120.207} C_DIS
LIN {X -0.005,Y -547.281,Z 775.462,A 0.000,B 0.000,C 90.000,E1 119.077} C_DIS
LIN {X 0.004,Y -549.996,Z 775.457,A 0.000,B 0.000,C 90.000,E1 118.231} C_DIS
LIN {X 0.044,Y -552.579,Z 775.452,A 0.000,B 0.000,C 90.000,E1 117.385} C_DIS
LIN {X 0.106,Y -554.790,Z 775.448,A 0.000,B 0.000,C 90.000,E1 116.539} C_DIS
LIN {X -0.056,Y -556.602,Z 775.443,A 0.000,B 0.000,C 90.000,E1 115.720} C_DIS
LIN {X -0.195,Y -558.159,Z 775.438,A 0.000,B 0.000,C 90.000,E1 114.899} C_DIS
LIN {X 0.193,Y -559.448,Z 775.434,A 0.000,B 0.000,C 90.000,E1 114.027} C_DIS
LIN {X 0.082,Y -561.821,Z 775.423,A 0.000,B 0.000,C 90.000,E1 112.099} C_DIS
LIN {X 0.307,Y -563.070,Z 775.417,A 0.000,B 0.000,C 90.000,E1 110.972} C_DIS
LIN {X 0.259,Y -564.727,Z 775.408,A 0.000,B 0.000,C 90.000,E1 109.322} C_DIS
LIN {X -0.203,Y -565.482,Z 775.403,A 0.000,B 0.000,C 90.000,E1 108.544} C_DIS
LIN {X -0.005,Y -566.605,Z 775.395,A 0.000,B 0.000,C 90.000,E1 107.149} C_DIS
LIN {X -0.174,Y -568.150,Z 775.385,A 0.000,B 0.000,C 90.000,E1 105.245} C_DIS
LIN {X -0.075,Y -569.505,Z 775.375,A 0.000,B 0.000,C 90.000,E1 103.592} C_DIS
LIN {X -0.250,Y -571.427,Z 775.363,A 0.000,B 0.000,C 90.000,E1 101.422} C_DIS
LIN {X -0.217,Y -572.851,Z 775.354,A 0.000,B 0.000,C 90.000,E1 99.782} C_DIS
LIN {X 0.018,Y -573.984,Z 775.347,A 0.000,B 0.000,C 90.000,E1 98.398} C_DIS
LIN {X -0.284,Y -575.067,Z 775.339,A 0.000,B 0.000,C 90.000,E1 97.068} C_DIS
LIN {X 0.001,Y -575.977,Z 775.332,A 0.000,B 0.000,C 90.000,E1 95.682} C_DIS
LIN {X 0.005,Y -577.175,Z 775.321,A 0.000,B 0.000,C 90.000,E1 93.784} C_DIS
LIN {X 0.229,Y -577.944,Z 775.314,A 0.000,B 0.000,C 90.000,E1 92.407} C_DIS
LIN {X 0.146,Y -578.372,Z 775.309,A 0.000,B 0.000,C 90.000,E1 91.604} C_DIS
LIN {X -0.040,Y -579.120,Z 775.300,A 0.000,B 0.000,C 90.000,E1 90.000} C_DIS
LIN {X 0.039,Y -579.556,Z 775.294,A 0.000,B 0.000,C 90.000,E1 88.912} C_DIS
LIN {X -0.112,Y -580.092,Z 775.285,A 0.000,B 0.000,C 90.000,E1 87.306} C_DIS
LIN {X -0.218,Y -580.534,Z 775.276,A 0.000,B 0.000,C 90.000,E1 85.698} C_DIS
LIN {X 0.258,Y -580.869,Z 775.267,A 0.000,B 0.000,C 90.000,E1 84.033} C_DIS
LIN {X -0.145,Y -581.107,Z 775.257,A 0.000,B 0.000,C 90.000,E1 82.186} C_DIS
LIN {X -0.019,Y -581.224,Z 775.248,A 0.000,B 0.000,C 90.000,E1 80.557} C_DIS
LIN {X 0.228,Y -581.277,Z 775.242,A 0.000,B 0.000,C 90.000,E1 79.454} C_DIS
LIN {X -0.104,Y -581.240,Z 775.236,A 0.000,B 0.000,C 90.000,E1 78.409} C_DIS
LIN {X 0.130,Y -581.043,Z 775.227,A 0.000,B 0.000,C 90.000,E1 76.769} C_DIS
LIN {X -0.072,Y -580.591,Z 775.218,A 0.000,B 0.000,C 90.000,E1 75.172} C_DIS
LIN {X 0.217,Y -580.148,Z 775.210,A 0.000,B 0.000,C 90.000,E1 73.795} C_DIS
LIN {X -0.221,Y -579.700,Z 775.203,A 0.000,B 0.000,C 90.000,E1 72.489} C_DIS
LIN {X -0.121,Y -578.970,Z 775.194,A 0.000,B 0.000,C 90.000,E1 70.859} C_DIS
LIN {X -0.227,Y -578.262,Z 775.186,A 0.000,B 0.000,C 90.000,E1 69.518} C_DIS
LIN {X -0.137,Y -577.425,Z 775.179,A 0.000,B 0.000,C 90.000,E1 68.156} C_DIS
LIN {X 0.096,Y -576.618,Z 775.173,A 0.000,B 0.000,C 90.000,E1 67.050} C_DIS
LIN {X -0.138,Y -575.506,Z 775.165,A 0.000,B 0.000,C 90.000,E1 65.717} C_DIS
LIN {X 0.293,Y -574.487,Z 775.159,A 0.000,B 0.000,C 90.000,E1 64.588} C_DIS
LIN {X 0.185,Y -573.298,Z 775.153,A 0.000,B 0.000,C 90.000,E1 63.512} C_DIS
LIN {X 0.050,Y -571.934,Z 775.147,A 0.000,B 0.000,C 90.000,E1 62.436} C_DIS
LIN {X 0.257,Y -569.952,Z 775.139,A 0.000,B 0.000,C 90.000,E1 61.051} C_DIS
LIN {X -0.160,Y -567.997,Z 775.133,A 0.000,B 0.000,C 90.000,E1 59.999} C_DIS
LIN {X 0.067,Y -566.397,Z 775.129,A 0.000,B 0.000,C 90.000,E1 59.154} C_DIS
LIN {X 0.081,Y -564.615,Z 775.124,A 0.000,B 0.000,C 90.000,E1 58.329} C_DIS
LIN {X -0.121,Y -561.927,Z 775.118,A 0.000,B 0.000,C 90.000,E1 57.248} C_DIS
LIN {X -0.143,Y -559.661,Z 775.113,A 0.000,B 0.000,C 90.000,E1 56.421} C_DIS
LIN {X -0.105,Y -556.335,Z 775.107,A 0.000,B 0.000,C 90.000,E1 55.308} C_DIS
LIN {X -0.189,Y -553.572,Z 775.103,A 0.000,B 0.000,C 90.000,E1 54.482} C_DIS
LIN {X -0.049,Y -551.589,Z 775.100,A 0.000,B 0.000,C 90.000,E1 53.909} C_DIS
LIN {X 0.137,Y -548.201,Z 775.095,A 0.000,B 0.000,C 90.000,E1 53.050} C_DIS
LIN {X 0.096,Y -545.141,Z 775.091,A 0.000,B 0.000,C 90.000,E1 52.351} C_DIS
LIN {X -0.072,Y -541.774,Z 775.087,A 0.000,B 0.000,C 90.000,E1 51.662} C_DIS
LIN {X -0.021,Y -538.934,Z 775.084,A 0.000,B 0.000,C 90.000,E1 51.090} C_DIS
LIN {X 0.178,Y -534.944,Z 775.080,A 0.000,B 0.000,C 90.000,E1 50.356} C_DIS
LIN {X -0.237,Y -531.416,Z 775.077,A 0.000,B 0.000,C 90.000,E1 49.828} C_DIS
LIN {X 0.076,Y -527.534,Z 775.074,A 0.000,B 0.000,C 90.000,E1 49.218} C_DIS
LIN {X 0.009,Y -523.107,Z 775.070,A 0.000,B 0.000,C 90.000,E1 48.647} C_DIS
LIN {X -0.136,Y -518.222,Z 775.067,A 0.000,B 0.000,C 90.000,E1 48.081} C_DIS
LIN {X 0.199,Y -514.517,Z 775.065,A 0.000,B 0.000,C 90.000,E1 47.634} C_DIS
LIN {X -0.226,Y -509.271,Z 775.062,A 0.000,B 0.000,C 90.000,E1 47.148} C_DIS
LIN {X -0.077,Y -503.406,Z 775.059,A 0.000,B 0.000,C 90.000,E1 46.581} C_DIS
LIN {X -0.254,Y -498.895,Z 775.057,A 0.000,B 0.000,C 90.000,E1 46.215} C_DIS
LIN {X -0.295,Y -492.806,Z 775.054,A 0.000,B 0.000,C 90.000,E1 45.729} C_DIS
LIN {X -0.235,Y -486.551,Z 775.051,A 0.000,B 0.000,C 90.000,E1 45.243} C_DIS
LIN {X -0.228,Y -478.592,Z 775.048,A 0.000,B 0.000,C 90.000,E1 44.676} C_DIS
LIN {X 0.144,Y -467.305,Z 775.044,A 0.000,B 0.000,C 90.000,E1 43.866} C_DIS
LIN {X -0.200,Y -447.848,Z 775.037,A 0.000,B 0.000,C 90.000,E1 42.609} C_DIS
LIN {X -0.264,Y -427.006,Z 775.028,A 0.000,B 0.000,C 90.000,E1 41.148} C_DIS
LIN {X 0.179,Y -416.149,Z 775.024,A 0.000,B 0.000,C 90.000,E1 40.253} C_DIS
LIN {X 0.038,Y -411.537,Z 775.022,A 0.000,B 0.000,C 90.000,E1 39.886} C_DIS
LIN {X 0.179,Y -407.550,Z 775.020,A 0.000,B 0.000,C 90.000,E1 39.483} C_DIS
LIN {X 0.149,Y -407.532,Z 775.020,A 0.000,B 0.000,C 90.000,E1 39.483} C_DIS
LIN {X -0.178,Y -405.581,Z 775.013,A 0.000,B 0.000,C 90.000,E1 38.382} C_DIS
LIN {X -0.088,Y -397.926,Z 774.992,A 0.000,B 0.000,C 90.000,E1 34.532} C_DIS
LIN {X -0.115,Y -397.922,Z 774.988,A 0.000,B 0.000,C 90.000,E1 33.833} C_DIS
LIN {X 0.008,Y -398.671,Z 774.972,A 0.000,B 0.000,C 90.000,E1 31.003} C_DIS
LIN {X 0.112,Y -399.904,Z 774.957,A 0.000,B 0.000,C 90.000,E1 28.180} C_DIS
LIN {X 0.176,Y -401.327,Z 774.943,A 0.000,B 0.000,C 90.000,E1 25.720} C_DIS
LIN {X 0.086,Y -403.501,Z 774.926,A 0.000,B 0.000,C 90.000,E1 22.589} C_DIS
LIN {X -0.019,Y -407.152,Z 774.904,A 0.000,B 0.000,C 90.000,E1 18.779} C_DIS
LIN {X 0.172,Y -412.138,Z 774.883,A 0.000,B 0.000,C 90.000,E1 14.954} C_DIS
LIN {X -0.102,Y -415.827,Z 774.870,A 0.000,B 0.000,C 90.000,E1 12.591} C_DIS
LIN {X -0.108,Y -419.264,Z 774.859,A 0.000,B 0.000,C 90.000,E1 10.546} C_DIS
LIN {X -0.109,Y -422.740,Z 774.847,A 0.000,B 0.000,C 90.000,E1 8.511} C_DIS
LIN {X -0.181,Y -425.635,Z 774.838,A 0.000,B 0.000,C 90.000,E1 6.834} C_DIS
LIN {X -0.031,Y -430.355,Z 774.823,A 0.000,B 0.000,C 90.000,E1 4.131} C_DIS
LIN {X 0.152,Y -434.772,Z 774.810,A 0.000,B 0.000,C 90.000,E1 1.776} C_DIS
LIN {X -0.164,Y -439.368,Z 774.797,A 0.000,B 0.000,C 90.000,E1 359.484} C_DIS
LIN {X -0.057,Y -444.955,Z 774.782,A 0.000,B 0.000,C 90.000,E1 356.846} C_DIS
LIN {X 0.116,Y -450.219,Z 774.770,A 0.000,B 0.000,C 90.000,E1 354.546} C_DIS
LIN {X 0.105,Y -454.007,Z 774.761,A 0.000,B 0.000,C 90.000,E1 352.932} C_DIS
LIN {X 0.158,Y -457.735,Z 774.752,A 0.000,B 0.000,C 90.000,E1 351.319} C_DIS
LIN {X 0.175,Y -460.612,Z 774.745,A 0.000,B 0.000,C 90.000,E1 350.038} C_DIS
LIN {X -0.213,Y -463.348,Z 774.738,A 0.000,B 0.000,C 90.000,E1 348.814} C_DIS
LIN {X -0.207,Y -466.938,Z 774.729,A 0.000,B 0.000,C 90.000,E1 347.229} C_DIS
LIN {X -0.137,Y -468.711,Z 774.725,A 0.000,B 0.000,C 90.000,E1 346.589} C_DIS
LIN {X 0.054,Y -470.993,Z 774.722,A 0.000,B 0.000,C 90.000,E1 345.936} C_DIS
LIN {X 0.072,Y -473.354,Z 774.719,A 0.000,B 0.000,C 90.000,E1 345.463} C_DIS
LIN {X 0.101,Y -476.552,Z 774.717,A 0.000,B 0.000,C 90.000,E1 344.991} C_DIS
LIN {X 0.154,Y -479.699,Z 774.715,A 0.000,B 0.000,C 90.000,E1 344.629} C_DIS
LIN {X -0.190,Y -485.020,Z 774.712,A 0.000,B 0.000,C 90.000,E1 344.157} C_DIS
LIN {X 0.188,Y -493.449,Z 774.708,A 0.000,B 0.000,C 90.000,E1 343.449} C_DIS
LIN {X -0.171,Y -512.274,Z 774.701,A 0.000,B 0.000,C 90.000,E1 342.181} C_DIS
LIN {X -0.106,Y -528.101,Z 774.695,A 0.000,B 0.000,C 90.000,E1 341.148} C_DIS
LIN {X 0.094,Y -534.396,Z 774.693,A 0.000,B 0.000,C 90.000,E1 340.732} C_DIS
END
